# B&R Automation Studio project NewPendant_NG4_11_05_25A (part 22)

##### ArcLink.h
```c
#ifndef _ARCLINK_H
#define _ARCLINK_H

#include <bur/plctypes.h>

#include <runtime.h>

#include <..\..\Lib\utilityLib\bgdebug.h>

#include <..\..\Lib\utilityLib\libRingBuffer.h>

#include <..\..\Lib\arclink\NetworkActions.h>
#include <..\..\Lib\arclink\NetworkAttribute.h>
#include <..\..\Lib\arclink\ArcLinkObject.h>
#include <..\..\Lib\arclink\Robot.h>

#include <..\..\Lib\arclink\WeldController.h>
#include <..\..\Lib\arclink\NetworkBlocks.h>
#include <..\..\Lib\arclink\Attribute.h>

//#include <..\Lib\utilityLib\bgdebug.h>

/*

#include <..\Lib\utilityLib\libRingBuffer.h>

#include <..\Lib\arclink\NetworkActions.h>
#include <..\Lib\arclink\NetworkAttribute.h>
#include <..\Lib\arclink\ArcLinkObject.h>
#include <..\Lib\arclink\Robot.h>

#include <..\Lib\arclink\WeldController.h>
#include <..\Lib\arclink\NetworkBlocks.h>
#include <..\Lib\arclink\Attribute.h>

*/

#define ARC_LINK_OBJECT_BUS_MASTER_ADDRESS 	0
#define ARC_LINK_HEADER_SIZE 				10
#define ARC_LINK_REQUEST_SIZE 				18 // Without Data
#define ARC_LINK_RESPONSE_SIZE 				6 // Without Data

#define ARC_LINK_TXT_BUF_LEN 	512
#define ARC_LINK_TXT_REC_NUM 	8
#define ARC_LINK_TELEMETRY_DESTINATION_ADDRESS 128
#define ACR_LINK_TELEMETRY_ALL_OBJECT_ADDRESS 254

/* Arclink Message  */
typedef struct Arc_Link_Internal_typ{
	UDINT MaxMsgDataLength;
	USINT *pInMsg;
	UDINT  InMsgLen;
	USINT *pOutMsg;
	UDINT  OutMsgLen;

	USINT  InMsgCnt;
	USINT  OutMsgCnt;

} Arc_Link_Internal_typ;

/**
 * @author Obed Bardales
 *         <p>
 *         <b>ArcLink UDP Message Header</b>, which is required in any
 *         ArcLink/XT transmission, has the following structure:
 *         </p>
 *         <br>
 *
 */
typedef struct Arc_Link_Header_typ
{
		/**
	 * <b>Flags</b>: The Flags are a number of boolean settings which control
	 * the type and behavior of the given message packet. (See Table 13 2
	 * Message Header Flags Bit fields) <br>
	 * <b>Value / Range</b>: 0 to 65535 <br>
	 * <b>Size</b>: 2 <i>bytes</i><br>
	 * Bits Description<br>
	 * 0 (LSB) If not set, then the accompanying message is a request. If set,
	 * then the message is a response.<br>
	 * 1 If not set, then the accompanying message is a Server Command. If set,
	 * then the message is an ArcLink Command. ArcLink/XT does not use server
	 * commands; this bit must be set.<br>
	 * 2 Flag for whether Group Addressing is to be used. ArcLink/XT does not
	 * support Group requests; this bit must be cleared.<br>
	 * 3 Flag for whether Sessions should be used. ArcLink/XT does not use
	 * sessions; this bit must be cleared<br>
	 * 13 – 15 3-bit number (0 – 7) indicating the Last Error Type (to accompany
	 * LastError in the Message Header) (See Table 13 3 Error Types) <br>
	 * Table 13 2 Message Header Flags Bit fields <br>
	 * <br>
	 * Error Types<br>
	 * Type Description<br>
	 * 1 Port Error. Occurs in the event of a timeout or a framing error on a
	 * certain port.<br>
	 * 2 NA<br>
	 * 3 Windows Error. Occurs when a COM port fails, or on file access
	 * errors.<br>
	 * 4 Server Error. Occurs in the event of a timeout on the server side, a
	 * malformed ALTCP message, or a bad argument in a server command.<br>
	 * 5 ArcLink Error. Occurs on the ArcLink side only.<br>
	 * 6 WinSock Error. Occurs when a socket is closed unexpectedly. <br>
	 * Table 13 3 Error Types<br>
	 *
	 *
	 */
	UINT Flags;
	/**
	* <b>Sequence</b>: A simple number used to identify the process which
	* initially sent the request. Response should match request. Should not be
	* advanced on a message retry attempt. <br>
	* <b>Value / Range</b>: 0 to 65535 <br>
	* <b>Size</b>: 2 <i>bytes</i>
	*/
	UINT Sequence;
	/**
	 * <b>Last Error</b>: In responses, used to inform the application that an
	 * error occurred while processing the requested command. A value of 0
	 * implies no error. <br>
	 * <b>Value / Range</b>: 0 to 4G<br>
	 * <b>Size</b>: 4 <i>bytes</i>
	 */
	UDINT LastError;
	/**
	* <b>Data Length</b>: The size of the entire message packet, not including
	* this header. <br>
	* <b>Value / Range</b>: 0 to 65535<br>
	* <b>Size</b>: 2 <i>bytes</i>
	*/
	UINT DataLength;
} Arc_Link_Header_typ;

/*
	ArcLink ServiceID
*/
typedef struct ServiceID_typ{
	UINT 	AttributeNumber;
	USINT	StateNumber;
	USINT	PropertyNumber;
} ServiceID_typ;

/**
 * @author Obed Bardales
 *         <p>
 *         <b>ArcLink Requests</b>, If the incoming message is an ArcLink
 *         Command (Bit 1 of the Flags is set), then the data immediately
 *         following the header will be an ArcLink Command Request.
 *         </p>
 *         <br>
 *
 */
typedef struct Arc_Link_Request_typ
{
	/**
	 * <b>Timeout Time (10-ms ticks)</b>: Response time-out time for proxied CAN
	 * requests (default is 100), 20ms recommended.<br>
	 * <b>Value / Range</b>: 0 to 65535 <br>
	 * <b>Size</b>: 2 <i>bytes</i>
	 */
	UINT TimeoutTime;
	/**
	 * <b>Flags</b>: Several boolean settings to further configure the command
	 * request. (See Table 13.5 ArcLink Command Request Flags Bit fields)<br>
	 * <b>Value / Range</b>: 0 to 255 <br>
	 * <b>Size</b>: 1 <i>byte</i> Bits Description <br>
	 * (LSB) 0 - 1 Response Filter Type (0 to 3)<br>
	 * 0 = Match (default)<br>
	 * 1 = First-in<br>
	 * 2 Abort (default is false)<br>
	 * 3 Specifies whether the Timeout Time in the Command Request applies to
	 * each individual response (true) or all responses at once (false).<br>
	 *
	 */
	USINT Flags;
	/**
	 * <b>Retries</b>: Number of retry attempts for proxied CAN requests
	 * (default is 1)<br>
	 * <b>Value / Range</b>: 0 to 255 <br>
	 * <b>Size</b>: 1 <i>byte</i>
	 */
	USINT Retries;

	/**
	 * <b>Message Counter</b>: A simple number used to identify the process
	 * which initially sent the request. Response should match request. Should
	 * not be advanced on a message retry attempt. <br>
	 * <b>Value / Range</b>: 0 to 255 <br>
	 * <b>Size</b>: 1 <i>byte</i>
	 */
	USINT MessageCounter;

	/**
	 * <b>Addressing Mode</b>: Addressing Mode to use (default is peer-peer)
	 * (See Table 13 6 Addressing Modes) ArcLink/XT may not make requests using
	 * group addressing. <br>
	 * <b>Value / Range</b>: 0 to 255 <br>
	 * <b>Size</b>: 1 <i>byte</i><br>
	 * Mode Description <br>
	 * 0 Master-Slave<br>
	 * 1 Master-Slaves<br>
	 * 4 Slave-Master<br>
	 * 6 Peer-Peer<br>
	 * 7 Peer-Peers<br>
	 *
	 */
	USINT AddressingMode;

	/**
	 * <b>Connection ID</b>: Connection ID to use (default is 15) (See Table
	 * 13.7 Connection IDs) <br>
	 * <b>Value / Range</b>: 0 to 255 <br>
	 * <b>Size</b>: 1 <i>byte</i><br>
	 * ID Description<br>
	 * 2 Active Master-Slave<br>
	 * 3 Active Slave-Master Active Peer-Peer<br>
	 * 15 General<br>
	 *
	 */
	USINT ConnectionID;

	/**
	 * <b>Maximum Objs</b>: Maximum number of ArcLink Object respondents. If
	 * Group Addressing is not used, then this value must be set to 1.
	 * ArcLink/XT should set this field to 1. <br>
	 * <b>Value / Range</b>: 0 to 255 <br>
	 * <b>Size</b>: 1 <i>byte</i>
	 */
	USINT MaximumObjs;

	/**
	 * <b>Service ID</b>: (See Attribute Service ID)<br>
	 * <b>Value / Range</b>: ... <br>
	 * <b>Size</b>: 4 <i>bytes</i><br>
	 *
	 * Attributes are referenced using an attribute service ID. Table 15 2 shows
	 * that this structure includes an attribute number, a property number and a
	 * state number. The state is only relevant for attributes whose Attribute
	 * Class Property is set to 10 or 11, in which case the state field selects
	 * the state. If a state is not applicable for the attribute in question,
	 * the value in this field is ignored.<br>
	 *
	 * |Attribute Number| State Number |Attribute Property Number E.g. Value, Low limit, High limit| <br>
	 * |2 bytes |1 byte |1 byte |<br>
	 * Table 15 2- Attribute Service ID
	 *
	 *
	 */
	ServiceID_typ ServiceID;

	/**
	 * <b>Source Address</b>: Source address of the message.<br>
	 * <b>Value / Range</b>: 0 - 255 <br>
	 * <b>Size</b>: 1 <i>byte</i>
	 */
	USINT SourceAddress;

	/**
	 * <b>Destination Address</b>: Destination Address of the message. Either an
	 * ArcLink Object network address or an ArcLink Group Network address,
	 * depending on the Addressing Mode ArcLink/XT may not make requests using
	 * group addressing. <br>
	 * <b>Value / Range</b>: 0 - 255 <br>
	 * <b>Size</b>: 1 <i>byte</i><br>
	 *
	 * <b>24. ArcLink Object Classes</b><br>
	 * Object Object Class Function<br>
	 * Bus Master (BM) 0 Assigns (“maps”) ArcLink addresses.<br>
	 * Weld-Controller (WC) 1 Contains power on/off and welding process
	 * adjustments for the welding power supply.<br>
	 * Wire Drive (WD) 2 Contains motor on/off and set wire feed speed command
	 * value.<br>
	 * User Interface 3 Manual user interface<br>
	 * Gas Controller (GC) 4 Contains the gas on/off command to control the gas
	 * solenoid.<br>
	 * Sense Lead (SL) 5 Controls remote torch voltage electrode sense
	 * connection<br>
	 * DeviceNet Gateway 6 DeviceNet Gateway<br>
	 * Reserved 7 <br>
	 * Ethernet Gateway (GW) 8 Ethernet Gateway. This is the gateway over which
	 * ArcLink/XT messages arrive.<br>
	 * Spool Gun 9 Spool Gun<br>
	 * Robot 10 Controls the other objects.<br>
	 * Phase Generator 11 Phase Generator. In ACDC systems, this determines the
	 * frequency and phase relationships (from arc to arc).<br>
	 * Arc Object 12 The Arc Object is used in previous generation ACDC
	 * systems.<br>
	 * Reserved 13 <br>
	 * Dual User Interface 14 Dual manual feeder user interface.<br>
	 * Pendent 15 Manual operator pendent.<br>
	 * Reserved 16 <br>
	 * Process Monitor 17 The Process Monitor object records welding data and
	 * enforces process limits (if set).<br>
	 * Spread Arc 18 The spread arc device oscillates the welding torch.<br>
	 * Flux Hopper 19 The flux hopper dispenses flux in SAW welding.<br>
	 * Tractor Travel 20 The tractor moves the welding torch.<br>
	 * Travel Carriage 21 The travel carriage moves the welding torch.<br>
	 * Remote 22 The remote reads analog inputs (for remote analog
	 * pendants).<br>
	 * Stick/TIG UI 23 The Stick/TIG UI is a limited function manual user
	 * interface.<br>
	 * STT Switch 24 The STT switch is used in the STT process.<br>
	 * AC Switch 25 The AC switch is used in AC processes.<br>
	 *
	 */
	USINT DestinationAddress;

	/**
	 * <b>Service</b>: Number of the service to execute (See Appendix: Network
	 * Services) <br>
	 * <b>Value / Range</b>: 0 - 255 <br>
	 * <b>Size</b>: 1 <i>byte</i>
	 */
	USINT Service;

	/**
	 * <b>Max Response Size</b>: Maximum size of the response (in bytes) <br>
	 * <b>Value / Range</b>: 0 - 254 <br>
	 * <b>Size</b>: 1 <i>byte</i>
	 */
	USINT MaxResponseSize;

	/**
	 * <b>Request Size</b>: Size of outgoing ArcLink Data<br>
	 * <b>Value / Range</b>: 0 - 255 <br>
	 * <b>Size</b>: 1 <i>byte</i>
	 */
	USINT RequestSize;

	/**
	 * <b>Reserved</b>: A reserved byte<br>
	 * <b>Value / Range</b>: 0 - 255 <br>
	 * <b>Size</b>: 1 <i>byte</i>
	 */
	USINT Reserved;

	/**
	 * <b>OutgoingData</b>: Outgoing ArcLink data<br>
	 * <b>Value / Range</b>: ... <br>
	 * <b>Size</b>: 2+ <i>bytes</i>
	 */

	USINT* OutgoingData;
} Arc_Link_Request_typ;

/**
 * @author Obed Bardales
 *         <p>
 *         <b>ArcLink Response</b>, A response to an ArcLink Command request
 *         coming back from the machine must be preceded by an ALTCP header, as
 *         specified above. The header’s Flags must have bits 0 and 1 set to
 *         True in order to be identified as an ArcLink response. Immediately
 *         after the header, the ArcLink Command Response is structured as
 *         follows
 *         </p>
 *         <br>
 *
 */
typedef struct Arc_Link_Response_typ
{
	/**
	 * <b>Object Count</b>: Number of objects that responded to the ArcLink
	 * request<br>
	 * <b>Value / Range</b>: 0 to 255 <br>
	 * <b>Size</b>: 1 <i>byte</i>
	 */
	USINT ObjectCount;
	/**
	* <b>Reserved</b>: A reserved byte<br>
	* <b>Value / Range</b>: 0 to 255 <br>
	* <b>Size</b>: 1 <i>byte</i>
	*/
	USINT Reserved;
	/**
	 * <b>Status</b>: If the request had caused an ArcLink error, the error will
	 * be recorded in this status byte. If there was no error, status will be
	 * 0.<br>
	 * <b>Value / Range</b>: 0 to 255 <br>
	 * <b>Size</b>: 1 <i>byte</i>
	 */
	USINT Status;
	/**
	 * <b>Object Address</b>: The ArcLink network address of the object that
	 * responded. <br>
	 * <b>Value / Range</b>: 0 to 255 <br>
	 * <b>Size</b>: 1 <i>byte</i>
	 */
	USINT ObjectAddress;
	/**
	 * <b>Response Size</b>: The size (in bytes) of the incoming ArcLink Data
	 * <br>
	 * <b>Value / Range</b>: 0 to 254 <br>
	 * <b>Size</b>: 1 <i>byte</i>
	 */
	USINT ResponseSize;
	/**
	 * <b>Reserved</b>: A reserved byte<br>
	 * <b>Value / Range</b>: 0 to 255 <br>
	 * <b>Size</b>: 1 <i>byte</i>
	 */
	USINT Reserved2;
	/**
	 * <b>Response Data</b>: Incoming ArcLink Data<br>
	 * <b>Value / Range</b>: ... <br>
	 * <b>Size</b>: 2+ <i>bytes</i>
	 */
	USINT* ResponseData;
} Arc_Link_Response_typ;

/* Arclink Message  */
typedef struct Arc_Link_Message_typ{
	Arc_Link_Header_typ header;
	Arc_Link_Request_typ request;
	Arc_Link_Response_typ response;
} Arc_Link_Message_typ;

typedef struct PendingResponse_typ{
	BOOL WriteAttribute30770;   //1 Enable
	BOOL WriteAttribute30781;   //1 Enable
	BOOL WriteAttribute30758;   //1 Enable
	BOOL WriteAttribute30;
	BOOL CreateReadyReport;
	BOOL CreateFaultReport;

	UINT fsSequence;  // Sequence tracked for attribute 30731 (fault status)
	UINT sqConfigDataSearchAction;
	UINT sqReadCoolerSens;
	UINT WriteAttribute30770Sequence;
	UINT WriteAttribute30781Sequence;
	UINT WriteAttribute30758Sequence;
	UINT WriteAttribute30Sequence;
	UINT CreateReadyReportSequence;
	UINT CreateFaultReportSequence;
	UINT CreateReadControlParamDataAction;
	UINT sqConfigDataSearchAction_GasSol;

} PendingResponse_typ;

typedef struct Arc_Link_typ
{
	RingBuffer *bufIN; 		// Incoming Messages RingBuffer pointer
	RingBuffer *bufOUT; 	// Outgoing Messages RingBuffer pointer
	Arc_Link_Message_typ msgIN;		// Placeholder
	Arc_Link_Message_typ msgOUT;	// Placeholder
	Arc_Link_Internal_typ internal; // Internal
	Robot_typ robot; // Robot reference to this plc
	PendingResponse_typ PendingResponse; // pending response
} Arc_Link_typ;

/* Prototypes */
void ArcLink_cyclic(Arc_Link_typ *arc);
void ArcLink_init(Arc_Link_typ *arc , RingBuffer *bufIN, RingBuffer *bufOUT , UDINT  pInMsg  , UDINT  pOutMsg , UDINT recLen );

//////////////////////////////////////////////////////////////////////
// ArcLink Event Codes
// The following table lists the event codes that can be logged in Event Log postings
//////////////////////////////////////////////////////////////////////
#define	ARC_LINK_EVENT_11	11	/* 	Internal request failed to generate a response */
#define	ARC_LINK_EVENT_12	12	/* 	Internal attribute read/write failed */
#define	ARC_LINK_EVENT_13	13	/* 	Values/settings saved in the system could not be restored (corrupt)*/
#define	ARC_LINK_EVENT_14	14	/* 	Values/settings saved in the system could not be restored (primary section) */
#define	ARC_LINK_EVENT_15	15	/* 	Values/settings saved in the system could not be restored (secondary section) */
#define	ARC_LINK_EVENT_16	16	/* 	Values/settings that are saved could not be restored during powerup */
#define	ARC_LINK_EVENT_17	17	/* 	Serial port communication timed out*/
#define	ARC_LINK_EVENT_18	18	/* 	ArcLink auto-mapping failed*/
#define	ARC_LINK_EVENT_19	19	/* 	Excessive EEPROM saves detected for a certain attribute */
#define	ARC_LINK_EVENT_21	21	/* 	Device that controls sequence of the welding operation halted due to an error*/
#define	ARC_LINK_EVENT_22	22	/* 	Device that controls the sequence of the welding operation halted due to an error response when it tried to update a device's settings*/
#define	ARC_LINK_EVENT_23	23	/* 	Weld Sequencer could not change settings on a controlled object during welding*/
#define	ARC_LINK_EVENT_24	24	/* 	Error occurred while the weld sequencer was changing the weld mode*/
#define	ARC_LINK_EVENT_25	25	/* 	When updating non-state memory attributes via sequencer action, allow all but mode changing*/
#define	ARC_LINK_EVENT_26	26	/* 	Problem with paired mapping*/
#define	ARC_LINK_EVENT_27	27	/* 	Read/write request failed during paired mapping*/
#define	ARC_LINK_EVENT_28	28	/* 	Output locked out in the Weld Controller*/
#define	ARC_LINK_EVENT_29	29	/* 	Low-level DSP main control routine could not complete all of its tasks in time*/
#define	ARC_LINK_EVENT_31	31	/* 	Actual input current exceeded the input current limit*/
#define	ARC_LINK_EVENT_32	32	/* 	Capacitor bank A fell below the low voltage limit*/
#define	ARC_LINK_EVENT_33	33	/* 	Capacitor bank B fell below the low voltage limit*/
#define	ARC_LINK_EVENT_34	34	/* 	Capacitor bank A exceeded the high voltage limit*/
#define	ARC_LINK_EVENT_35	35	/* 	Capacitor bank B exceeded the high voltage limit*/
#define	ARC_LINK_EVENT_36	36	/* 	System detected a temperature level beyond the normal system operating limit*/
#define	ARC_LINK_EVENT_37	37	/* 	System failed to initialize inverter hardware during startup*/
#define	ARC_LINK_EVENT_38	38	/* 	Momentary AC dropout*/
#define	ARC_LINK_EVENT_39	39	/* 	Miscellaneous hardware fault occurred whose source cannot be determined*/
#define	ARC_LINK_EVENT_41	41	/* 	Long-term average secondary (weld) current limit has been exceeded*/
#define	ARC_LINK_EVENT_42	42	/* 	System detected a ground fault has occurred*/
#define	ARC_LINK_EVENT_43	43	/* 	Voltage difference between Capacitor bank A and B was greater than the allowable limit*/
#define	ARC_LINK_EVENT_44	44	/* 	Main processor in the system did not respond to another processor within the allotted time*/
#define	ARC_LINK_EVENT_45	45	/* 	Welding voltage was above limit*/
#define	ARC_LINK_EVENT_46	46	/* 	Output amperage limit exceeded*/
#define	ARC_LINK_EVENT_47	47	/* 	Miscellaneous hardware fault (capacitor fault or heart beat fault)*/
#define	ARC_LINK_EVENT_48	48	/* 	Miscellaneous hardware fault (main contactor open)*/
#define	ARC_LINK_EVENT_49	49	/* 	Single phase input operation has been detected*/
#define	ARC_LINK_EVENT_51	51	/* 	Weld Controller failed to set weld sequencer schedule memory*/
#define	ARC_LINK_EVENT_52	52	/* 	Digital Signal Processor (DSP) in the system is no longer responding to heartbeat request from the main processor*/
#define	ARC_LINK_EVENT_53	53	/* 	System detected the loss of a voltage sense lead*/
#define	ARC_LINK_EVENT_54	54	/* 	Long-term average secondary (weld) current limit has been exceeded*/
#define	ARC_LINK_EVENT_55	55	/* 	Communication with DSP failed*/
#define	ARC_LINK_EVENT_56	56	/* 	Communication with Chopper failed*/
#define	ARC_LINK_EVENT_57	57	/* 	Function Generator reported an error*/
#define	ARC_LINK_EVENT_58	58	/* 	Primary input power board not ready*/
#define	ARC_LINK_EVENT_59	59	/* 	Reduced input power detected*/
#define	ARC_LINK_EVENT_61	61	/* 	Step value for either upslope or downslope was calculated to zero*/
#define	ARC_LINK_EVENT_62	62	/* 	Weld Sequencer did not get a positive response after sending out Weld Cycle Data twice*/
#define	ARC_LINK_EVENT_63	63	/* 	Problem with submerged arc Slave device*/
#define	ARC_LINK_EVENT_71	71	/* 	Secondary over-power*/
#define	ARC_LINK_EVENT_72	72	/* 	Unsupported hardware revision*/
#define	ARC_LINK_EVENT_81	81	/* 	Feed head experienced a motor overload fault*/
#define	ARC_LINK_EVENT_82	82	/* 	Feed head experienced a motor over current fault*/
#define	ARC_LINK_EVENT_83	83	/* 	Wire drive shutdown bit 1 circuit open*/
#define	ARC_LINK_EVENT_84	84	/* 	Wire drive shutdown bit 2 circuit open (Water Fault)*/
#define	ARC_LINK_EVENT_85	85	/* 	Object could not find the Arc Control Object to send the I/O trigger command*/
#define	ARC_LINK_EVENT_86	86	/* 	Wire Drive input voltage too high*/
#define	ARC_LINK_EVENT_87	87	/* 	Wire Drive failed to find another object*/
#define	ARC_LINK_EVENT_88	88	/* 	Wire Drive could not send the trigger to the specified object in the event data.*/
#define	ARC_LINK_EVENT_89	89	/* 	Wire Drive failed to find the Production Monitoring object for profile selection based on digital inputs*/
#define	ARC_LINK_EVENT_91	91	/* 	Sense Lead object could not update the weld sequencer's or the weld controller's polarity attribute.*/
#define	ARC_LINK_EVENT_92	92	/* 	Remote shutdown of Weld Controller*/
#define	ARC_LINK_EVENT_95	95	/* 	Spool Gun shutdown due to motor drawing excessive current*/
#define	ARC_LINK_EVENT_96	96	/* 	Weld Controller failed to read WFS decimal places*/

//////////////////////////////////////////////////////////////////////
// ArcLink Error Codes
// The following table lists the event codes that can be logged in Event Log postings
//////////////////////////////////////////////////////////////////////
#define	ARC_LINK_ERROR_0	0	/*	Success (no message error). */
#define	ARC_LINK_ERROR_1  	1	/*	Attribute not found. */
#define ARC_LINK_ERROR_2	2	/* 	Attribute value is read-only. */
#define ARC_LINK_ERROR_3	3 	/* 	Attribute Value (being written) is out of limits.*/
#define ARC_LINK_ERROR_4	4	/* 	Attribute Value (being written) is above high limit.*/
#define ARC_LINK_ERROR_5	5	/* 	Attribute Value (being written) is below low limit.*/
#define ARC_LINK_ERROR_8	8	/*	ArcLink object not found (bad ArcLink object address).*/
#define ARC_LINK_ERROR_9	9	/*	Attribute property specified is invalid.*/
#define ARC_LINK_ERROR_11	11	/*	Attribute property is not applicable (e.g. units code for Boolean type).  Only while reading.*/
#define ARC_LINK_ERROR_12	12	/*	Attribute property is not supported (e.g. invalid type id, or not applicable).  For reads or writes.*/
#define ARC_LINK_ERROR_13	13	/*	Attribute property is read-only.*/
#define ARC_LINK_ERROR_14	14	/*	Attribute is invalid.*/
#define ARC_LINK_ERROR_15	15	/*	ArcLink Object messages could not be relayed over Ethernet.*/
#define ARC_LINK_ERROR_16 	16	/*	ArcLink service busy (message should be re-sent).*/
#define ARC_LINK_ERROR_17	17	/*	ArcLink service busy (message should be re-sent).*/
#define ARC_LINK_ERROR_18	18	/*	ArcLink service busy (message should be re-sent).*/
#define ARC_LINK_ERROR_20	20	/*	ArcLink Block ID not found (for block read or write service).*/
#define ARC_LINK_ERROR_21	21	/*	ArcLink Action ID not found (for action service).*/
#define ARC_LINK_ERROR_22	22	/*	ArcLink Group Address not found.*/
#define ARC_LINK_ERROR_23	23	/*	ArcLink Event ID not found.*/
#define ARC_LINK_ERROR_24	24	/*	ArcLink Service not supported.*/
#define ARC_LINK_ERROR_25	25	/*	ArcLink Service not available.*/
#define ARC_LINK_ERROR_26	26	/*	Fragment buffer busy (message should be re-sent).*/
#define ARC_LINK_ERROR_27	27	/*	Fragment out of sequence (message should be re-started).*/
#define ARC_LINK_ERROR_28	28	/*	Fragment receive time out (message should be re-started).*/
#define ARC_LINK_ERROR_29	29	/*	Fragment message invalid.*/
#define ARC_LINK_ERROR_30	30	/*	Message request size is invalid.*/
#define ARC_LINK_ERROR_31	31	/*	Message response buffer was too small.*/
#define ARC_LINK_ERROR_33	33	/*	Message time out (message should be re-started).*/
#define ARC_LINK_ERROR_34	34	/*	Write failed.*/
#define ARC_LINK_ERROR_35	35	/*	Read failed.*/
#define	ARC_LINK_ERROR_36	36	/*	Invalid selection.*/
#define	ARC_LINK_ERROR_37	37	/*	ArcLink Object was busy (message should be re-sent). */

//////////////////////////////////////////////////////////////////////
// Attribute Value Property ID Codes
//////////////////////////////////////////////////////////////////////
/*
 * Value 0 Defined by Attribute Data Type
 */
#define PROPERTY_ID_VALUE 0

/**
 * Class 1 Unsigned Int (1)
 */
#define PROPERTY_ID_CLASS 1

/**
 * Saved In E2 2 Boolean
 */
#define PROPERTY_ID_SAVED_IN_E2 2

/**
 * Attribute Data Type 3 Unsigned Int (1)
 */
#define PROPERTY_ID_ATTRIBUTE_DATA_TYPE 3

/**
 * Unit Code 4 Unsigned Int (1)
 */
#define PROPERTY_ID_UNIT_CODE 4

/**
 * High Limit 5 Defined by Attribute Data Type
 */
#define PROPERTY_ID_HIGH_LIMIT 5

/**
 * Low Limit 6 Defined by Attribute Data Type
 */
#define PROPERTY_ID_LOW_LIMIT 6

/**
 * Decimal Places 7 Unsigned Int (1)
 */
#define PROPERTY_ID_DECIMAL_PLACES 7

/**
 * Name 8 String (1-254)
 */
#define PROPERTY_ID_NAME 8

//////////////////////////////////////////////////////////////////////
// Attribute Data Type Property, ID Codes
//////////////////////////////////////////////////////////////////////
/**
 * <b>Boolean</b>:<br>
 * <i>size: 1 byte</i>
 */
#define DATA_TYPE_BOOLEAN 0

/**
 * <b>Enumerated 1</b>:<br>
 * <i>size: 1 byte</i>
 */
#define DATA_TYPE_ENUMERATED_1 1

/**
 * <b>Enumerated 2</b>:<br>
 * <i>size: 2 bytes</i>
 */
#define DATA_TYPE_ENUMERATED_2 2

/**
 * <b>Enumerated 4</b>:<br>
 * <i>size: 4 bytes</i>
 */
#define DATA_TYPE_ENUMERATED_4 3

/**
 * <b>Bit Mapped 1</b>:<br>
 * <i>size: 1 byte</i>
 */
#define DATA_TYPE_BIT_MAPPED_1 4

/**
 * <b>Bit Mapped 2</b>:<br>
 * <i>size: 2 bytes</i>
 */
#define DATA_TYPE_BIT_MAPPED_2 5

/**
 * <b>Bit Mapped 4</b>:<br>
 * <i>size: 4 bytes</i>
 */
#define DATA_TYPE_BIT_MAPPED_4 6

/**
 * <b>Signed Integer 1</b>:<br>
 * <i>size: 1 byte</i>
 */
#define DATA_TYPE_SIGNED_INTEGER_1 7

/**
 * <b>Signed Integer 2</b>:<br>
 * <i>size: 2 bytes</i>
 */
#define DATA_TYPE_SIGNED_INTEGER_2 8

/**
 * <b>Signed Integer 4</b>:<br>
 * <i>size: 4 bytes</i>
 */
#define DATA_TYPE_SIGNED_INTEGER_4 9

/**
 * <b>Unsigned Integer 1</b>:<br>
 * <i>size: 1 byte</i>
 */
#define DATA_TYPE_UNSIGNED_INTEGER_1 10

/**
 * <b>Unsigned Integer 2</b>:<br>
 * <i>size: 2 bytes</i>
 */
#define DATA_TYPE_UNSIGNED_INTEGER_2 11

/**
 * <b>Unsigned Integer 4</b>:<br>
 * <i>size: 4 bytes</i>
 */
#define DATA_TYPE_UNSIGNED_INTEGER_4 12

/**
 * <b>Floating Point</b>:<br>
 * <i>size: 4 bytes</i>
 */
#define DATA_TYPE_FLOATING_POINT 13

/**
 * <b>ASCII String </b>:<br>
 * <i>size: (0 - 254) bytes</i>
 */
#define DATA_TYPE_ASCII_STRING 14

//////////////////////////////////////////////////////////////////////
// Attribute Class Codes
//////////////////////////////////////////////////////////////////////
/**
 * <b>Network Configuration</b>:<br>
 * Inputs related to the network. E.g. Group Assignment <br>
 *
 */
#define CLASS_NETWORK_CONFIGURATION 0

/**
 * <b>Network Status</b>:<br>
 * Outputs describing information related to the network. E.g. Network
 * Version Number <br>
 * <i>Read Only</i>
 */
#define CLASS_NETWORK_STATUS 1

/**
 * <b>Command</b>:<br>
 * Inputs used to activate an object?s behavior. Changes generally have an
 * immediate effect. E.g. Gas Purge<br>
 *
 */
#define CLASS_COMMAND 2

/**
 * <b>Reference</b>:<br>
 * Inputs which are set points. Changes generally have an immediate effect.
 * E.g. Cold Inch<br>
 *
 */
#define CLASS_REFERENCE 3

/**
 * <b>Reference</b>:<br>
 * Inputs which alter the object?s general behavior. E.g. Motor Control-Loop
 * Mode<br>
 *
 */
#define CLASS_CONFIGURATION 4

/**
 * <b>Signal</b>:<br>
 * Outputs used for metering and monitoring. E.g. Actual Arc Current <br>
 * <i>Read Only</i>
 */
#define CLASS_SIGNAL 5

/**
 * <b>Status</b>:<br>
 * Outputs used for metering and monitoring. E.g. Faults<br>
 * <i>Read Only</i>
 */
#define CLASS_STATUS 6

/**
 * <b>Sequence Controlled Command</b>:<br>
 * Command to be controlled by the Sequencer object (object class 0). E.g.
 * Motor On/Off<br>
 */
#define CLASS_SEQUENCE_CONTROLLED_COMMAND 7

/**
 * <b>Sequence Controlled Reference</b>:<br>
 * Reference to be controlled by the Sequencer object (object class 0). E.g.
 * Commanded WFS<br>
 */
#define CLASS_SEQUENCE_CONTROLLED_REFERENCE 8

/**
 * <b>Sequence Controlled Configuration</b>:<br>
 * Configuration to be controlled by the Sequencer object (object class 0).
 * E.g. Weld Procedure <br>
 */
#define CLASS_SEQUENCE_CONTROLLED_CONFIGURATION 9

/**
 * <b>Command with State Memory</b>:<br>
 * Command which has state memory. The sequencer object creates attributes
 * of this class from attributes of class 7. The state portion of the
 * service ID is relevant for the read and write services.<br>
 */
#define CLASS_COMMAND_WITH_STATE_MEMORY 10

/**
 * <b>Reference with State Memory</b>:<br>
 * Reference which has state memory. The sequencer object creates attributes
 * of this class from attributes of class 8. The state portion of the
 * service ID is relevant for the read and write services.<br>
 */
#define CLASS_REFERENCE_WITH_STATE_MEMORY 11

/**
 * <b>Debug</b>:<br>
 * Used (primarily) during manufacturing.
 */
#define CLASS_DEBUG 12

/**
 * <b>Setup</b>:<br>
 */
#define CLASS_SETUP 13

/**
 * <b>Version</b>:<br>
 * Version related information.<br>
 * <i>Read Only</i>
 */
#define CLASS_VERSION 14

//////////////////////////////////////////////////////////////////////
// Addresing mode
//////////////////////////////////////////////////////////////////////
#define ADDRESS_MODE_MASTER_SLAVE	 0
#define ADDRESS_MODE_MASTER_SLAVES	 1
#define ADDRESS_MODE_SLAVE_MASTER	 4
#define ADDRESS_MODE_PEER_PEER		 6
#define ADDRESS_MODE_PEER_PEERS 	 7

//////////////////////////////////////////////////////////////////////
// Network Services Codes
//////////////////////////////////////////////////////////////////////
/**
 * <b>Attribute Read</b>:<br>
 */
#define NETWORK_SERVICE_ATTRIBUTE_READ 0

/**
 * <b>Attribute Write</b>:<br>
 */
#define NETWORK_SERVICE_ATTRIBUTE_WRITE 1

/**
 * <b>Confirmed Event Report</b>:<br>
 */
#define NETWORK_SERVICE_CONFIRMED_EVENT_REPORT 2

/**
 * <b>Unconfirmed Event Report</b>:<br>
 */
#define NETWORK_SERVICE_UNCONFIRMED_EVENT_REPORT 3

/**
 * <b>Action</b>:<br>
 */
#define NETWORK_SERVICE_ACTION 4

/**
 * <b>Read Block</b>:<br>
 */
#define NETWORK_SERVICE_READ_BLOCK 5

/**
 * <b>Write Block</b>:<br>
 */
#define NETWORK_SERVICE_WRITE_BLOCK 6

/**
 * <b>Confirmed Event Block Report</b>:<br>
 */
#define NETWORK_SERVICE_CONFIRMED_EVENT_BLOCK_REPORT 7

/**
 * <b>Unconfirmed Event Block Report</b>:<br>
 */
#define NETWORK_SERVICE_UNCONFIRMED_EVENT_BLOCK_REPORT 8

//#include <..\..\Lib\arclink\Handler.h>

#endif /* _ARCLINK_H */
```

##### Robot.c
```c
/*
 * Handler.c
 *
 *  Created on: May 18, 2017
 *      Author: Obed Bardales
 */
#ifndef _ROBOT_C
#define _ROBOT_C

/* Handle Robot Cyclic Operations */
void handleRobotCyclicOps(Arc_Link_typ *arc){
	if(!arc) return;

	// Handle Mr.Robot interface
	handleRobotInterface(arc);

	// "The difference is not one thing, it's everything!"
}

/* Get Network Configuration from Robot */
void getNetworkConfigurationAttribute(Arc_Link_typ *arc, USINT *ResponseData){
	Arc_Link_Request_typ *req;
	Arc_Link_Response_typ *r;
	Robot_typ *robot;
	ServiceID_typ *serviceID;
	ArcLinkObject_typ *arclink;
	USINT data[10]; // Temp Data place holder
	UINT txtlength; // text length

	if(!arc) return;
	if(!ResponseData) return;

	robot = &arc->robot; // Reference to Robot
	req = &arc->msgIN.request;
	serviceID = &req->ServiceID;
	r = &arc->msgOUT.response;
	arclink = &robot->arclink;
	int dataSize = req->MaxResponseSize;

	/* Attribute Number */
	switch (serviceID->AttributeNumber) {

		case VENDOR_ID: /* 0 */
			// MaxDataSize = 2
			// Big Endian Format

			data[0] = (USINT) (arclink->network.VendorID >> 8);
			data[1] = (USINT) (arclink->network.VendorID >> 0);
			memcpy(ResponseData, data, 2);
			r->ResponseSize = 2;

			return;

		case CLASS_ID: /* 4 */
			// MaxDataSize = 2
			// Big Endian Format
			data[0] = (USINT) (arclink->network.ClassID >> 8);
			data[1] = (USINT) (arclink->network.ClassID >> 0);
			memcpy(ResponseData, data, 2);
			r->ResponseSize = 2;
			return;

		case CLASS_TYPE: /* 7 */
			// MaxDataSize = 2
			// Big Endian Format
			data[0] = (USINT) (arclink->network.ClassType >> 0);
			memcpy(ResponseData, data, 1);
			r->ResponseSize = 1;
			return;

		case GROUP_ASSIGNMENTS: /* 10 */
			// MaxDataSize = 2
			// Big Endian Format
			data[0] = (USINT) (arclink->network.GroupAssignments >> 0);
			memcpy(ResponseData, data, 1);
			r->ResponseSize = 1;
			return;

		case INSTANCE_ASSIGNMENTS: /* 11 */
			// MaxDataSize = 2
			// Big Endian Format
			data[0] = (USINT) (arclink->network.InstanceAssignments >> 0);
			memcpy(ResponseData, data, 1);
			r->ResponseSize = 1;
			return;

		case FAULT_STATUS: /* 14 */
			// MaxDataSize = 2
			// Big Endian Format
			data[0] = (USINT) (arclink->network.FaultStatus >> 0);
			memcpy(ResponseData, data, 1);
			r->ResponseSize = 1;
			return;

		case SILICON_SERIAL_NUMBER: /* 16 */
			// MaxDataSize = 2
			// Big Endian Format
			data[0] = (USINT) (arclink->network.SiliconSerialNumber >> 8);
			data[1] = (USINT) (arclink->network.SiliconSerialNumber >> 0);
			memcpy(ResponseData, data, 2);
			r->ResponseSize = 2;
			return;

		case NUMBER_OF_EMBEDDED_OBJECTS: /* 17 */
			// MaxDataSize = 2
			// Big Endian Format
			data[0] = (USINT) (arclink->network.NumberofEmbeddedObjects >> 0);
			memcpy(ResponseData, data, 1);
			r->ResponseSize = 1;
			return;

		case SOFTWARE_VERSION: /* 19 */
			// MaxDataSize = 64
			// Big Endian Format
			txtlength = strlen(arclink->network.SoftwareVersion);
			// Swap Bytes before sendSuccesfullWriteAttributeConfirmation
			//swapBytes(arclink->network.SoftwareVersion, txtlength);
			memcpy(ResponseData, arclink->network.SoftwareVersion, txtlength);
			//swapBytes(arclink->network.SoftwareVersion, txtlength);
			r->ResponseSize = txtlength;
			return;

		case BOOTSTRAP: /* 24 */
			// MaxDataSize = 2
			// Big Endian Format
			data[0] = (USINT) (arclink->network.Bootstrap >> 0);
			memcpy(ResponseData, data, 1);
			r->ResponseSize = 1;
			return;

		case PAIRED_ITEMS_COUNT: /* 50 */
			// MaxDataSize = 2
			// Big Endia Format
			data[0] = (USINT) (arclink->network.PairedItemsCount >> 8);
			data[1] = (USINT) (arclink->network.PairedItemsCount >> 0);
			memcpy(ResponseData, data, 2);
			r->ResponseSize = 2;
			return;
	}
}

/* Write Network Configuration Attribute */
BOOL writeNetworkConfigurationAttribute(Arc_Link_typ *arc){

	BOOL success = 1;

	UINT *data;

	Arc_Link_Request_typ *req;
	ServiceID_typ *serviceID;
	Robot_typ *robot;
	ArcLinkObject_typ *arclink;
	if(!arc) return;

	req = &arc->msgIN.request;
	serviceID = &req->ServiceID;
	robot = &arc->robot;
	arclink = &robot->arclink;

	DBG("Inside writeNetworkConfigurationAttribute \r\n" );
	//Log.d(TAG, "Recevied Assign Network Address Action");

	// Copy Data if available to the Incoming data pointer
	if(req->RequestSize > 0){
	//byte[] data = r.OutgoingData; // incominng data in Big endian format
		data = (arc->internal.pInMsg + ARC_LINK_HEADER_SIZE + ARC_LINK_REQUEST_SIZE); // Pointer to data
	}else{
		DBG("Error: writeNetworkConfigurationAttribute, Error with Request size\r\n" );
		return;
	}

	/* Attribute Number */
	switch (serviceID->AttributeNumber) {

	// Currently Supported Attributes by the Robot
	case RESET:
		arclink->network.Reset = *(data + 0);//data[0]; // Size is typically 1 byte
		arclink->network.BusAvailable = 0; // Robot must enter to unmapped state
		robot->isMapping = 0;
		robot->isMapped = 0;
		robot->Cntrl.Fbk.Status &= ~ArcLink_Mapped;
		robot->Cntrl.Fbk.Status &= ~ArcLink_Mapping;
		robot->isMiscSetupOneShot = 0;
		DBG("Setting Robot to Unmapped state\r\n" );
		break;

	case GROUP_ASSIGNMENTS:
		arclink->network.GroupAssignments = *(data + 0);///data[0]; // Size is typically 1
													// byte

		break;

	case INSTANCE_ASSIGNMENTS:
		arclink->network.InstanceAssignments = *(data + 0);///data[0]; // Size is typically
														// 1 byte
		break;

	case BUS_AVAILABLE:
		arclink->network.BusAvailable = *(data + 0); //data[0]; // Size is typically 1 byte
		robot->isMapping 	= 0;
		robot->isMapped 	= 1;
		robot->Cntrl.Fbk.Status |= ArcLink_Mapped;
		robot->Cntrl.Fbk.Status &= ~ArcLink_Mapping;
		DBG("Robot was mapped succesfully Świetny programista! \r\n" );
		log_event(&robot->eventlog , "Arc Link Mapped");
		break;

	}

	return success; // Whether Attribute was written succesfully

}

void handleRobotInterface(Arc_Link_typ *arc){

	Robot_typ *robot;
	Robot_Intrf_typ *intrf;
	if(!arc) return;

	robot = &arc->robot;
	intrf = &robot->Intrf;

	// Robot must be Mapped with WeldController
	if(!robot->isMapped) return;

	//  Handle state changes from outside and provide feedback

	handleRobotCntrl(arc);
	error_status_handler(arc);
	ArcLink_Timer(arc);
	/////////

	// Handle xCMD
	switch(intrf->xCMD) {
		/* Turn Power Supply ON */
		case ROBOT_CMD_PS_ON:
			writeOutputOnCommand(arc);
			DBG("Robot commanded Power Supply ON! \r\n" );
			log_event(&robot->eventlog , "PS ON Cmd");
			break;

		/* Turn Power Supply OFF */
		case ROBOT_CMD_PS_OFF:
			writeOutputOffCommand(arc);
			DBG("Robot commanded Power Supply OFF! \r\n" );
			log_event(&robot->eventlog , "PS OFF Cmd");
			break;

		/* Set Controls Action Request */
		case ROBOT_SET_CONTROLS:
			createSetControlsAction(arc);
			DBG("Robot sent Set Controls Action Request! \r\n" );
			break;

		case ROBOT_CMD_COOLER_ON:
			writeOutputCoolerOnCommand(arc);
			DBG("Robot commanded Cooler ON! \r\n" );

		break;

		case ROBOT_CMD_COOLER_OFF:
			writeOutputCoolerOffCommand(arc);
			DBG("Robot commanded Cooler OFF! \r\n" );

		break;

		case ROBOT_CMD_SEARCH_COOLER_ADR:
			action_ConfigDataSearch_Cooler(arc);
			DBG("commanded Get Cooler Adr! \r\n" );
		break;

		case ROBOT_READ_COOLER_SENS:
			readAttribute_CoolerSens(arc);
			DBG("commanded Get Cooler Sens! \r\n" );
		break;

		case ROBOT_READ_WC_PARAM_DATA:
			createReadCntrlParamDataAction(arc);
			DBG("commanded Read WC Param Data! \r\n" );
		break;

		case ROBOT_CMD_SEARCH_GAS_SOL_ADR:
			action_ConfigDataSearch_GasSol(arc);
			DBG("commanded Get Gas Sol  Adr! \r\n" );
		break;

		case ROBOT_CMD_GAS_SOL_ENABLE: // Make  Gas Sol “Manual Valve”

			writeOutputGasEnableCommand(arc);
			DBG("Robot commanded Gas Enable\r\n" );

		break;

		case ROBOT_CMD_GAS_SOL_ON: // Turn On Gas Sol

			writeOutputGasOnCommand(arc);
			DBG("Robot commanded Gas ON\r\n" );

		break;

		case ROBOT_CMD_GAS_SOL_OFF:	// Turn Off Gas Sol

			writeOutputGasOffCommand(arc);
			DBG("Robot commanded Gas OFF\r\n" );

		break;

	}

	// Clear xCMD
	if (intrf->xCMD > 0) intrf->xCMD = 0;

}

void handleRobotCntrl(Arc_Link_typ *arc){

	Robot_typ *robot;
	Robot_Intrf_typ *intrf;
	if(!arc) return;

	robot = &arc->robot;
	intrf = &robot->Intrf;

	//*************** CMD  *****************************/
	//**************Highest priority CMD****************//
	if(robot->Cntrl.Cmd.COOLER && !robot->Cntrl.Int._COOLER){

		intrf->xCMD = ROBOT_CMD_COOLER_ON;
		robot->Cntrl.Int._COOLER  = robot->Cntrl.Cmd.COOLER;

	}
	else if(robot->Cntrl.Cmd.RUN != robot->Cntrl.Int._RUN){

		if(robot->Cntrl.Cmd.RUN)
			intrf->xCMD = ROBOT_CMD_PS_ON;
		else
			intrf->xCMD = ROBOT_CMD_PS_OFF;

		robot->Cntrl.Int._RUN  = robot->Cntrl.Cmd.RUN;
	}
	else if(!robot->Cntrl.Cmd.COOLER && robot->Cntrl.Int._COOLER){

		intrf->xCMD = ROBOT_CMD_COOLER_OFF;
		robot->Cntrl.Int._COOLER  = robot->Cntrl.Cmd.COOLER;

	}
	//robot->Cntrl.Int._RUN  = robot->Cntrl.Cmd.RUN;
	//robot->Cntrl.Int._COOLER  = robot->Cntrl.Cmd.COOLER;

	//********************************************************//

	if(!intrf->xCMD){

		/*
		1 Byte	Parameter Mask
		2 Bytes	Weld Mode 	If parameter mask bit 0 set.
		2 Bytes	Work-point	If parameter mask bit 1 set.
		2 Bytes	Trim	If parameter mask bit 2 set.
		2 Bytes	Wave-Control 1	If parameter mask bit 3 set.
		2 Bytes	Wave-Control 2	If parameter mask bit 4 set.
		2 Bytes	Wave-Control 3	If parameter mask bit 5 set.
		2 Bytes	Wave-Control 4	If parameter mask bit 6 set.
		*/

		switch(robot->Cntrl.Cmd.Mode){

			case 3:

				if((robot->Cntrl.Cmd.Mode != robot->Cntrl.Int._Mode )
					|| (robot->Cntrl.Cmd.AmpSP != robot->Cntrl.Int._AmpSP )
					|| (robot->Cntrl.Cmd.BckAmpSP != robot->Cntrl.Int._BckAmpSP )
					|| (robot->Cntrl.Cmd.PulseFreq != robot->Cntrl.Int._PulseFreq )
					|| (robot->Cntrl.Cmd.PulseWidth != robot->Cntrl.Int._PulseWidth )){

					robot->wc.setup.ctrlParam.ParameterMask = 0x23; // 0b0100011; // change accordingly for Mode 3
					UINT *mode 	= &robot->Cntrl.Cmd.Mode; // Mode
					UINT ampSP = (UINT)robot->Cntrl.Cmd.AmpSP; //amps
					robot->wc.setup.ctrlParam.WeldMode = *mode;
					robot->wc.setup.ctrlParam.WorkPoint = ampSP;
					robot->wc.setup.ctrlParam.WaveControl3 = 1; // Hot pulse. Need info from Lincoln

					// This command write Controls Parameter into Power Supply
					intrf->xCMD = ROBOT_SET_CONTROLS;

				}

				robot->Cntrl.Int._Mode 			= robot->Cntrl.Cmd.Mode;
				robot->Cntrl.Int._AmpSP 		= robot->Cntrl.Cmd.AmpSP;
				robot->Cntrl.Int._BckAmpSP 		= robot->Cntrl.Cmd.BckAmpSP;
				robot->Cntrl.Int._PulseFreq 	= robot->Cntrl.Cmd.PulseFreq;
				robot->Cntrl.Int._PulseWidth 	= robot->Cntrl.Cmd.PulseWidth;

			break;

			case 5:

				if((robot->Cntrl.Cmd.Mode != robot->Cntrl.Int._Mode )
					|| (robot->Cntrl.Cmd.Volts != robot->Cntrl.Int._Volts )
					|| (robot->Cntrl.Cmd.Pinch != robot->Cntrl.Int._Pinch )
					){

					robot->wc.setup.ctrlParam.ParameterMask = 0x0D; // 0b0001011; // change accordingly for Mode 5
					UINT *mode 	= &robot->Cntrl.Cmd.Mode; // Mode
					UINT VoltsSP = (UINT)(robot->Cntrl.Cmd.Volts * 10); //Volts
					robot->wc.setup.ctrlParam.WeldMode = *mode;
					robot->wc.setup.ctrlParam.WorkPoint = VoltsSP;
					robot->wc.setup.ctrlParam.WaveControl1 = (UINT)(robot->Cntrl.Cmd.Pinch * 10);

					// This command write Controls Parameter into Power Supply
					intrf->xCMD = ROBOT_SET_CONTROLS;

				}

				robot->Cntrl.Int._Mode 			= robot->Cntrl.Cmd.Mode;
				robot->Cntrl.Int._Volts 		= robot->Cntrl.Cmd.Volts;
				robot->Cntrl.Int._Pinch 		= robot->Cntrl.Cmd.Pinch;

			break;

			case 21:

				if((robot->Cntrl.Cmd.Mode != robot->Cntrl.Int._Mode )
					|| (robot->Cntrl.Cmd.WFS != robot->Cntrl.Int._WFS)
					|| (robot->Cntrl.Cmd.Volts != robot->Cntrl.Int._Volts )
					|| (robot->Cntrl.Cmd.Pinch != robot->Cntrl.Int._Pinch )
					|| robot->Cntrl.Cmd.SendParam
					){

					robot->Cntrl.Cmd.SendParam = 0;

					robot->wc.setup.ctrlParam.ParameterMask = 0x0F; // 0b0001111; // change accordingly for Mode 5
					UINT *mode 	= &robot->Cntrl.Cmd.Mode; // Mode
					UINT WFS_SP = (UINT)(robot->Cntrl.Cmd.WFS * 1); //WF
					UINT VoltsSP = (UINT)(robot->Cntrl.Cmd.Volts * 10); //Volts
					UINT PinchSP = (UINT)(robot->Cntrl.Cmd.Pinch * 10); //Pinch

					if(robot->Cntrl.Cmd.Development)
						robot->wc.setup.ctrlParam.WeldMode = 0;
					else
						robot->wc.setup.ctrlParam.WeldMode = *mode;

					robot->wc.setup.ctrlParam.WorkPoint = WFS_SP;
					robot->wc.setup.ctrlParam.Trim = VoltsSP;
					robot->wc.setup.ctrlParam.WaveControl1 = PinchSP;

					// This command write Controls Parameter into Power Supply
					intrf->xCMD = ROBOT_SET_CONTROLS;

					robot->Cntrl.Int._Mode 			= robot->Cntrl.Cmd.Mode;
					robot->Cntrl.Int._WFS 			= robot->Cntrl.Cmd.WFS;
					robot->Cntrl.Int._Volts 		= robot->Cntrl.Cmd.Volts;
					robot->Cntrl.Int._Pinch 		= robot->Cntrl.Cmd.Pinch;

				}

			break;

			case 22:

				if((robot->Cntrl.Cmd.Mode != robot->Cntrl.Int._Mode )
					|| (robot->Cntrl.Cmd.WFS != robot->Cntrl.Int._WFS)
					|| (robot->Cntrl.Cmd.Trim != robot->Cntrl.Int._Trim )
					|| (robot->Cntrl.Cmd.UltimArc != robot->Cntrl.Int._UltimArc )
					|| robot->Cntrl.Cmd.SendParam
					){

					robot->Cntrl.Cmd.SendParam = 0;

					robot->wc.setup.ctrlParam.ParameterMask = 0x0F; // 0b0001111; // change accordingly for Mode 5
					UINT *mode 	= &robot->Cntrl.Cmd.Mode; // Mode
					UINT WFS_SP = (UINT)(robot->Cntrl.Cmd.WFS * 1); // WF
					UINT TrimSP = (UINT)(robot->Cntrl.Cmd.Trim * 100); // Trim
					UINT UltimArcSP = (UINT)(robot->Cntrl.Cmd.UltimArc * 10); //Pinch

					if(robot->Cntrl.Cmd.Development)
						robot->wc.setup.ctrlParam.WeldMode = 0;
					else
						robot->wc.setup.ctrlParam.WeldMode = *mode;

					robot->wc.setup.ctrlParam.WorkPoint = WFS_SP;
					robot->wc.setup.ctrlParam.Trim = TrimSP;
					robot->wc.setup.ctrlParam.WaveControl1 = UltimArcSP;

					// This command write Controls Parameter into Power Supply
					intrf->xCMD = ROBOT_SET_CONTROLS;

					robot->Cntrl.Int._Mode 			= robot->Cntrl.Cmd.Mode;
					robot->Cntrl.Int._WFS 			= robot->Cntrl.Cmd.WFS;
					robot->Cntrl.Int._Trim 			= robot->Cntrl.Cmd.Trim;
					robot->Cntrl.Int._UltimArc 		= robot->Cntrl.Cmd.UltimArc;

				}

			break;

			case 160:
			case 161:
			case 162:
			case 163:
			case 164:
			case 165:
			case 166:
			case 167:

				if((robot->Cntrl.Cmd.Mode != robot->Cntrl.Int._Mode )
					|| (robot->Cntrl.Cmd.Volts != robot->Cntrl.Int._Volts )
					//|| (robot->Cntrl.Cmd.Pinch != robot->Cntrl.Int._Pinch )
					){

					robot->wc.setup.ctrlParam.ParameterMask = 0x03; // 0b0000011; // Volts and WaveCntr 1

					//robot->wc.setup.ctrlParam.ParameterMask = 0x01; // Only Volts

					UINT *mode 	= &robot->Cntrl.Cmd.Mode; // Mode
					UINT VoltsSP = (UINT)(robot->Cntrl.Cmd.Volts * 10); // Volts
					robot->wc.setup.ctrlParam.WeldMode = *mode;
					robot->wc.setup.ctrlParam.WorkPoint = VoltsSP;
					//robot->wc.setup.ctrlParam.WaveControl1 = (UINT)(robot->Cntrl.Cmd.Pinch * 10);
					robot->wc.setup.ctrlParam.WaveControl1 = 0;

					// This command write Controls Parameter into Power Supply
					intrf->xCMD = ROBOT_SET_CONTROLS;

				}

				robot->Cntrl.Int._Mode 			= robot->Cntrl.Cmd.Mode;
				robot->Cntrl.Int._Volts 		= robot->Cntrl.Cmd.Volts;
				//robot->Cntrl.Int._Pinch 		= robot->Cntrl.Cmd.Pinch;

			break;

			case 170:

				if((robot->Cntrl.Cmd.Mode != robot->Cntrl.Int._Mode )
					|| (robot->Cntrl.Cmd.WFS != robot->Cntrl.Int._WFS)
					|| (robot->Cntrl.Cmd.Volts != robot->Cntrl.Int._Volts )
					|| (robot->Cntrl.Cmd.UltimArc != robot->Cntrl.Int._UltimArc )
					|| robot->Cntrl.Cmd.SendParam
					){

					robot->Cntrl.Cmd.SendParam = 0;

					robot->wc.setup.ctrlParam.ParameterMask = 0x0F; // 0b0001111; // change accordingly for Mode 5
					UINT *mode 	= &robot->Cntrl.Cmd.Mode; // Mode
					UINT WFS_SP = (UINT)(robot->Cntrl.Cmd.WFS * 1); //WF
					UINT VoltsSP = (UINT)(robot->Cntrl.Cmd.Volts * 10); //Volts
					UINT UltimArcSP = (UINT)(robot->Cntrl.Cmd.UltimArc * 10); //UltimArc

					if(robot->Cntrl.Cmd.Development)
						robot->wc.setup.ctrlParam.WeldMode = 0;
					else
						robot->wc.setup.ctrlParam.WeldMode = *mode;

					robot->wc.setup.ctrlParam.WorkPoint = WFS_SP;
					robot->wc.setup.ctrlParam.Trim = VoltsSP;
					robot->wc.setup.ctrlParam.WaveControl1 = UltimArcSP;

					// This command write Controls Parameter into Power Supply
					intrf->xCMD = ROBOT_SET_CONTROLS;

					robot->Cntrl.Int._Mode 			= robot->Cntrl.Cmd.Mode;
					robot->Cntrl.Int._WFS 			= robot->Cntrl.Cmd.WFS;
					robot->Cntrl.Int._Volts 		= robot->Cntrl.Cmd.Volts;
					robot->Cntrl.Int._UltimArc 		= robot->Cntrl.Cmd.UltimArc;

				}

			break;

			case 200:  // Calibration Current

				if((robot->Cntrl.Cmd.Mode != robot->Cntrl.Int._Mode )
					|| (robot->Cntrl.Cmd.AmpSP != robot->Cntrl.Int._AmpSP )
					){

					robot->wc.setup.ctrlParam.ParameterMask = 0x03; // 0b0000011; // change accordingly for Mode 200
					UINT *mode 	= &robot->Cntrl.Cmd.Mode; // Mode
					UINT AmpSP = (UINT)(robot->Cntrl.Cmd.AmpSP * 1); //amps
					robot->wc.setup.ctrlParam.WeldMode = *mode;
					robot->wc.setup.ctrlParam.WorkPoint = AmpSP;

					// This command write Controls Parameter into Power Supply
					intrf->xCMD = ROBOT_SET_CONTROLS;

				}

				robot->Cntrl.Int._Mode 			= robot->Cntrl.Cmd.Mode;
				robot->Cntrl.Int._AmpSP 		= robot->Cntrl.Cmd.AmpSP;

			break;

		}

	}
	//********************************************************//

	//*****************Lowest Priority CMD ********************//
	if(!intrf->xCMD){
		if(robot->Cntrl.Cmd.RST != robot->Cntrl.Int._RST){

			robot->Cntrl.Fbk.Status = 0;
			robot->miscSetup.state = 0; //reset misc state machine state
			robot->miscSetup.CoolerAddr = 0;
			robot->isMapping = 0;
			robot->isMapped = 0;	    //clear flag, set to unmapped status, stop timer
			robot->isMiscSetupOneShot = 0;
			robot->Comm.ArcComTimer.IN = 0;
			robot->Comm.StopRespondHeartBeat = 1; //halt heartbeat,force master to send out RESET request

		}
		robot->Cntrl.Int._RST 			= robot->Cntrl.Cmd.RST;

	}

	//*************** FEEDBACK  *****************************/

	robot->Cntrl.Fbk.curArcVolt = robot->wc.data.telemetry.fVoltage;
	robot->Cntrl.Fbk.curArcAmp  = robot->wc.data.telemetry.fCurrent;
	//robot->Cntrl.Fbk.Error      =  ???????
	//robot->Cntrl.Fbk.Status      =  ???????

	//********************************************************//

	return;

}

void error_status_handler(Arc_Link_typ *arc)
{

	Robot_typ *robot;
	if(!arc) return;

	robot = &arc->robot;

	// System is ready when mapped, ready status from PS is set and Arc Link Active, could add no system fault here
	if ((robot->isReady) && (robot->isMapped) && (robot->Comm.ArcLinkActive) && !robot->Cntrl.Fbk.Error)
	{
		robot->Cntrl.Fbk.Status |= PS_Ready;
//		log_event(&robot->eventlog , "Power supply is ready");
	}

	else
		robot->Cntrl.Fbk.Status &= ~PS_Ready;

	/*
	if ((robot->Cntrl.Fbk.Error >> 1 & 0x0001) || (robot->Cntrl.Fbk.Error >> 2 & 0x0001))  //either system fault from PS or network error will generate fault condition
		robot->Cntrl.Fbk.Error |= PS_Error_Present;
	else
		robot->Cntrl.Fbk.Error &= ~PS_Error_Present;
	*/
}
void ArcLink_Timer(Arc_Link_typ *arc){
//
	Robot_typ *robot;
	if(!arc) return;

	robot = &arc->robot;

	robot->Comm.PT = 2000; // 2s  timeout

	robot->Comm.CoolerSensPull_PT = 500; // 0.5s  timer

    robot->Comm.ArcComTimer.PT = robot->Comm.PT;

	if (robot->Comm.HeartBeat_Received && (robot->Comm.ArcComTimer.ET > 0)) //everytime got heartbeat, reset timer, to prevent trigger timeout
	    robot->Comm.ArcComTimer.IN = 0;

	else if (robot->Comm.HeartBeat_Received && (robot->Comm.ArcComTimer.ET == 0)){ //start timer, reset heartbeat flag
		if (robot->isMapped){  //
			robot->Comm.ArcComTimer.IN = 1;
		}
		if (robot->Comm.ClearError)    // clear error once getting connectivity from PS
		{
			robot->Comm.ClearError = 0;
			robot->Cntrl.Fbk.Error = 0;
			log_event(&robot->eventlog , "Network is active");
		}
		robot->Comm.HeartBeat_Received = 0;   //reset flag to start watchdog

	}

	TON(&robot->Comm.ArcComTimer);  //2 seconds Watchdog

    if (!robot->Comm.ArcComTimer.Q)
	robot->Comm.ArcLinkActive = 1;  // 1 Active
	else
	robot->Comm.ArcLinkActive = 0;	//timeout

	if (!robot->Comm.ArcLinkActive)
	{
		DBG_OB("Arc Link Disconnected\r\n");
		robot->Cntrl.Fbk.Error |= ArcLink_Com_Failed;
		robot->Cntrl.Fbk.Status = 0;
		robot->isMapping = 0;
		robot->isMapped = 0;	    //clear flag, set to unmapped status, stop timer
		robot->isMiscSetupOneShot = 0;
		robot->Comm.ArcComTimer.IN = 0;
		robot->Comm.ClearError = 1;	 //set flag when getting communication back, reset error
		log_event(&robot->eventlog , "Network is down");
	}
	else if (robot->isMapped)
	{
	/*	DBG_OB("Arc Link Connected\r\n"); */
		robot->Cntrl.Fbk.Error &= ~ArcLink_Com_Failed;
		robot->Cntrl.Fbk.Status |= ArcLink_Active;

	}

	// Pull Cooler Sens Status

	if((robot->miscSetup.CoolerAddr > 0)
		&& (robot->Comm.CoolerSensPull_PT > 0)){

		robot->Comm.CoolerSensPullTimer.PT = robot->Comm.CoolerSensPull_PT;

		if(robot->isMapped && robot->Comm.ArcLinkActive){

			if(!robot->Comm.CoolerSensPullTimer.IN){
				readAttribute_CoolerSens(arc);
				DBG("commanded Get Cooler Sens! \r\n" );
				robot->Comm.CoolerSensPullTimer.IN = 1;
				//TON(&robot->Comm.CoolerSensPullTimer);
			}
			else if(robot->Comm.CoolerSensPullTimer.Q){

				robot->Comm.CoolerSensPullTimer.IN = 0;
				//TON(&robot->Comm.CoolerSensPullTimer);

			}
			//else
				//TON(&robot->Comm.CoolerSensPullTimer);

		}

		TON(&robot->Comm.CoolerSensPullTimer);
	}

}
#endif /* _ROBOT_C */
```

### Program Logical/Libraries/bglibas

#### bgssm.c
```c
/********************************************************************
 * COPYRIGHT -- belgor
 ********************************************************************
 * Library: bglibas
 * File: bglibas.c
 * Author: admin
 * Created: March 07, 2012
 ********************************************************************
 * Implementation of library bglibas
 ********************************************************************/

#include <bur/plctypes.h>
#ifdef __cplusplus
	extern "C"
	{
#endif

	#include "bglibas.h"

#ifdef __cplusplus
	};
#endif

#include <string.h>

/* Init state machine. MUST be called once, before any other bgSSM function call. */
unsigned long bgSSMInit(struct bgSSM_typ* p, unsigned long pFunGetStateName, unsigned long pFunCyclicCallback)
{
	/*TODO: Add your code here*/
	memset(p, 0, sizeof(struct bgSSM_typ));

	p->pfunGetStateName = (UDINT)pFunGetStateName;
	p->pfunCyclicCallback = (UDINT)pFunCyclicCallback;
	p->stateInit = 1;
	return(0);
}
/* State machine cyclic operation. */
unsigned long bgSSMCyclic(struct bgSSM_typ* p)
{
	/*TODO: Add your code here*/
	int ii;

	//operate all timers
	for(ii=0; ii<BGSSM_TIMER_COUNT;ii++){
		bgTimerCyclic(&p->timer_x1ms[ii]);
	}
	bgTimerCyclic(&p->dlytimer_x1ms);

	//operate dlyCycle counter
	if(p->dlyCycles){
		p->dlyCycles--;
	}

	//call cyclic callback function if defined
	if(p->pfunCyclicCallback){
		void(*callback)(bgSSM_typ*) = ( void (*) (bgSSM_typ*) ) p->pfunCyclicCallback;
		(*callback)(p);
	}

	//clear single cycle flag every scan
	p->stateInit = 0;

	//check if state change requested
	if(p->state != p->stateNext){

		//if state change w. delay > wait for delay timer to expire or dlyCycles == 0
		if(!bgTimerIsTimeOut(&p->dlytimer_x1ms) || p->dlyCycles){
			return 1;
		}

		p->state = p->stateNext;
		//generate stateInit sigle scan flag
		p->stateInit = 1;

		//define state name if exteranl function for state names is defined
		if( p->pfunGetStateName ){
			char*(*getStateName)(UDINT) = ( char* (*) (UDINT) )p->pfunGetStateName;
			strcpy(p->stateText, (*getStateName)(p->state));
		}else{
			strcpy(p->stateText, "???");
		}
	}
	return(0);
}
/* Change to next state. */
unsigned long bgSSMStateNext(struct bgSSM_typ* p, unsigned long stateNext)
{
	/*TODO: Add your code here*/
	p->stateNext = stateNext;
	return(p->stateNext);
}

/* Change to next state w. timer delay. */
unsigned long bgSSMStateNextTimeDelay(struct bgSSM_typ* p, unsigned long stateNext, unsigned long delayTimeX1ms)
{
	/*TODO: Add your code here*/
	p->stateNext = stateNext;
	bgTimerStart(&p->dlytimer_x1ms, delayTimeX1ms);
	return(p->stateNext);
}

/* Change to next state w. cycles delay. */
unsigned long bgSSMStateNextCycleDelay(struct bgSSM_typ* p, unsigned long stateNext, unsigned long delayCycles)
{
	/*TODO: Add your code here*/
	p->stateNext = stateNext;
	p->dlyCycles = delayCycles;
	return(p->stateNext);
}
/* Check if first scan for the state. */
plcbit bgSSMIsStateInit(struct bgSSM_typ* p)
{
	/*TODO: Add your code here*/
	return(p->stateInit);
}
//EOF

/* Get current state */
unsigned long bgSSMGetState(struct bgSSM_typ* p)
{
	/*TODO: Add your code here*/
	return(p->state);
}

/* Get current state text*/
plcstring* bgSSMGetStateText(struct bgSSM_typ* p)
{
	/*TODO: Add your code here*/
	return(&p->stateText[0]);
}
```

- Library Logical/Libraries/sprintf2 (ANSIC) (no source held here)

### udpApp.var
```iecst
(********************************************************************
 * COPYRIGHT -- HP
 ********************************************************************
 * File: Global.var
 * Author: goran
 * Created: January 23, 2013
 ********************************************************************
 * Global variables of project YieldPlus
 ********************************************************************)
VAR
	gTxEvent : BOOL := FALSE;
	gTxRply : BOOL := FALSE;
	gJsontextTxRply : STRING[PAI_PVILIGHT_UDP_MSG_SIZE_MAX];
	gJsontextRx : STRING[PAI_PVILIGHT_UDP_MSG_SIZE_MAX];
	gJsontext : STRING[PAI_PVILIGHT_UDP_MSG_SIZE_MAX];
END_VAR
```

### cJSON.var
```iecst
(********************************************************************
 * COPYRIGHT -- HP
 ********************************************************************
 * Package: cJSON
 * File: cJSON.var
 * Author: goran
 * Created: June 19, 2013
 ********************************************************************
 * Variables of package cJSON
 ********************************************************************)
VAR
	gPaiPVILists : paiPVIListCollection_typ := (0);
	gHashValuesArray : ARRAY[0..19] OF UDINT;
	mHashCalcDone : UDINT;
	mHashCalcDlyTmr : TON;
END_VAR
```

### Program Logical/UDP/paiUDPService/udpclient

#### udpclient.c
```c
/********************************************************************
 * COPYRIGHT -- belgor
 ********************************************************************
 * Program: udpclient
 * File: udpclient.c
 * Author: goran
 * Created: January 23, 2013
 ********************************************************************
 * Implementation of program udpclient
 ********************************************************************/

#include <bur/plctypes.h>

#ifdef _DEFAULT_INCLUDES
	#include <AsDefault.h>
#endif

#include <../../../bglib/bgstring.c>
//#include <../../../bglib/bgTimer1ms.c>
//#include <string.h>

enum{
	udpCliZero = 0,
	udpCliInit,
	udpCliOpen,
	udpCliConnect,
	udpCliIdle,
	udpCliTxData,
	udpCliDisconnect,
	udpCliClose,
	udpCliError,
	udpCliLast
}STATEMACHINE;

static const char* udpCliStateName(int state)
{
static const char* stateNames[] = {
"Zero",
"Init",
"Open",
"Connect",
"Idle",
"TxData",
"Disconnect",
"Close",
"Error",
};

	if( state >= udpCliLast)
		return "unknow";

	return stateNames[state];
};

#define UDP_TX_BUF_SIZE_DEVICEDRIVER 100000
_LOCAL UDINT udpTxBufSize;

/*
###############################################################################
Utilities
###############################################################################
*/

static void convertIPTextToDigits(udpIPAddress_typ* p)
{
unsigned char txtbuffer[64];
bgStringList_typ list;

	strcpy((void*)txtbuffer, (void*)(p->text));
	list.src = txtbuffer;

	bgStringSplitLine(&list, '.');
	if(list.itemCount != 4){
		p->digit3 = 0;
		p->digit2 = 0;
		p->digit1 = 0;
		p->digit0 = 0;
		return;
	}
	p->digit3 = (USINT)atoi((UDINT)list.items[0]);
	p->digit2 = (USINT)atoi((UDINT)list.items[1]);
	p->digit1 = (USINT)atoi((UDINT)list.items[2]);
	p->digit0 = (USINT)atoi((UDINT)list.items[3]);
}

/**
 Simple logging
 Log goes to an array of PV strings > see _LOCAL STRING log[][] variable below
 Log output is visible via Automation Studio watch window
 Example of a log statement used within the code is:
 DBG(lgr, "This is log example. %d ", value1);
 To complety disable logging from this source file, change next line to: #if 0
*/
#if 1
#include <../../../bglib/bgPVLogger.c>
#define LOG_ENTRY_COUNT 20	//max number of log entries
#define LOG_ENTRY_LENGTH  32 //max length of individual log message. Longer msg are truncated
_LOCAL STRING log[LOG_ENTRY_COUNT][LOG_ENTRY_LENGTH]; //log output visible from Automation Studio!
static bgPVLogger_typ lgr;	//PV logger object
#else
#define DBG(loggerInstance, format, args...) ;
#define DBGINIT(loggerInstance, logoutput, logEntryCount, logEntrySize)  ;
#endif

/*
###############################################################################
Functions
###############################################################################
*/

static void udpClientSMCyclic(udpClient_typ *p)
{
bgSSM_typ* pSm = &p->sm;

	//operate timer(s)
	bgTimerCyclic(&pSm->timer_x1ms[0]); // delay timer

	//TimerExecute(&pSm->timer2x1ms); // update rate timer (in continues mode)
	//IMPORANT: for high speed, can't use TON block > rather, use cycle time
	if(pSm->timer_x1ms[1].ET)
		pSm->timer_x1ms[1].ET--;

	bgTimerCyclic(&pSm->timer_x1ms[2]); // 1sec stats timer

	//stats timers
	if( bgTimerIsTimeOut(&pSm->timer_x1ms[2]) ){
		bgTimerStart(&pSm->timer_x1ms[2], 1000);

		//values for cummulative (per min) calculations for datagrams
		p->txStats.datagramPerSec = pSm->counter[0];
		pSm->counter[0] = 0;
		if(p->txStats.datagramPerSec > p->txStats.datagramPerSecMax){
			p->txStats.datagramPerSecMax = p->txStats.datagramPerSec;
		}

		//values for cummulative (per min) calculations for bytes
		p->txStats.bytesPerSec = pSm->counter[1];
		pSm->counter[1] = 0;
		if(p->txStats.bytesPerSec > p->txStats.bytesPerSecMax){
			p->txStats.bytesPerSecMax = p->txStats.bytesPerSec;
		}
	}

	/*execute control state machine cyclic handler*/
	bgSSMCyclic(pSm);

	//show change of state in a log
	if( bgSSMIsStateInit(pSm) ){
		DBG(lgr, "sm=%s(%d)", bgSSMGetStateText(pSm), bgSSMGetState(pSm));
	}

	switch( bgSSMGetState(pSm) ){
		//========================================
		case udpCliZero:
			bgSSMStateNext(pSm, udpCliInit);
		break;
		//========================================
		case udpCliInit:
			if(p->clientIf.iConnect){
				bgSSMStateNext(pSm, udpCliOpen);
			}
		break;
		//========================================
		case udpCliOpen:

			if( bgSSMIsStateInit(pSm) ){
				p->client.open.enable = 1;
				p->client.open.port = 0;
				p->client.open.pIfAddr = 0;
//IMPORTANT:
//in order for the following conditional compilation to work properly, PLC object in the Configuration view
//must contain following defintion:
//Folder: Build
//Field: Additional Build Options
//Value: -D $(AS_CONFIGURATION)
//Using the above, name of the current AS configuration (i.e. realhw1 or testsim or else) becomes
//a defined preprocessor name. As a result, it's possible to destinguish between different configurations!
#ifdef Simulation
				//In case of testsim (ARsim) target, don't use socket options
				p->client.open.options = 0;
#warning "ISM Project - ARsim target!"
#else
				//For all other (real) targets, use socket options
				p->client.open.options = udpOPT_REUSEPORT | udpOPT_BROADCAST;
#warning "ISM Project - real target!"
#endif
				return;
			}

			if(p->client.open.status == ERR_FUB_BUSY)
				return;

			p->client.open.enable = 0;

			if(p->client.open.status == ERR_OK){
				p->client.recv.ident = p->client.open.ident;
				p->client.send.ident = p->client.open.ident;
				p->client.close.ident = p->client.open.ident;
				p->client.connect.ident = p->client.open.ident;
				p->client.disconnect.ident = p->client.open.ident;
				p->client.ioctl.ident = p->client.open.ident;

				udpTxBufSize = UDP_TX_BUF_SIZE_DEVICEDRIVER;
				p->client.ioctl.pData = &udpTxBufSize;
				p->client.ioctl.datalen = sizeof(udpTxBufSize);
				p->client.ioctl.ioctl = udpSO_SNDBUF_SET;
				p->client.ioctl.enable = 1;

				bgSSMStateNext(pSm, udpCliConnect);
				return;
			}

			DBG(lgr,"Err udp.open=%d", p->client.open.status);
			bgSSMStateNext(pSm, udpCliError);

		break;
		//========================================
		case udpCliConnect:

			if( bgSSMIsStateInit(pSm) ){
				p->client.connect.enable = 1;
				p->client.connect.port = p->clientIf.iRmtUdpPort;
				p->client.connect.pHost = (UDINT)p->clientIf.iRmtIPAddr;
				p->client.ioctl.enable = 0;
				return;
			}

			if(p->client.connect.status == ERR_FUB_BUSY)
				return;

			//p->client.connect.enable = 0;

			if(p->client.connect.status == ERR_OK){
				strcpy(p->clientIf.oRmtIpAddr, p->clientIf.iRmtIPAddr);
				p->clientIf.oRmtUdpPort = p->clientIf.iRmtUdpPort;

				bgSSMStateNext(pSm, udpCliIdle);
				return;
			}

			DBG(lgr,"Err udp.connect=%d", p->client.connect.status);
			bgSSMStateNext(pSm, udpCliError);

		break;
		//========================================
		case udpCliIdle:

			if( bgSSMIsStateInit(pSm) ){

			}

			if(!p->clientIf.iConnect){
				DBG(lgr,"disconnect request");
				bgSSMStateNext(pSm, udpCliDisconnect);
				return;
			}

			//udp client in echo mode!?
			//check for iSendEcho set by the server upon it receives a message > client sends out to the same host
			if((p->clientIf.iMode == 0) && p->clientIf.iSendEcho){
				p->clientIf.iSendEcho = 0;
				p->clientIf.iSend = 1;
				strcpy(p->clientIf.iRmtIPAddr, p->clientIf.iSendEchoRmtIpAddr);
			}

			//udp client in continues mode!?
			//trigger send update at a configured rate to a defined (sipplied to the inputs) remote host/port
			if(p->clientIf.iMode == 1){

				if(!pSm->timer_x1ms[1].ET){
					int updateTimeMs;

					if( p->clientIf.iUpdateRate ){
						updateTimeMs = 1000 /  p->clientIf.iUpdateRate;
					}else{
						updateTimeMs = 1000;
					}

					if(updateTimeMs < 10)
						updateTimeMs = 12;

					if(updateTimeMs > 1000)
						updateTimeMs = 1000;

					if(p->clientIf.iTaskCycleTimeXms){
						pSm->timer_x1ms[1].ET= updateTimeMs / p->clientIf.iTaskCycleTimeXms;
					}else{
						pSm->timer_x1ms[1].ET= updateTimeMs / gUdpClient_TaskCycleTimeXms; // devide by task clas time to find out increments
					}

					p->clientIf.iSend = 1;
				}
			}

			//monitor for change in remote host settings
			//in case of a change > reconnect (disconncet then connect)
			if((p->clientIf.oRmtUdpPort != p->clientIf.iRmtUdpPort) ||
				strcmp(p->clientIf.oRmtIpAddr, p->clientIf.iRmtIPAddr)
			){
				DBG(lgr,"rmt settings changed. Triggering reconnect.");
				bgSSMStateNext(pSm, udpCliDisconnect);
				return;
			}

			//monitor request to send
			if(!p->clientIf.iSend){
				return;
			}
			p->clientIf.iSend = 0;

			if(p->clientIf.iTxDataLen > UDP_CLIENT_TXBUF_SIZE){
				p->clientIf.iTxDataLen = UDP_CLIENT_TXBUF_SIZE;
			}

			if(!p->clientIf.iTxDataAdr && !p->clientIf.iTxCallback){
				DBG(lgr,"udp.send nothing to tx");
				return;
			}

			//execute memcpy if datasource is defined
			if(p->clientIf.iTxDataAdr){
				memcpy((void*)(p->txbuf), (void*)(p->clientIf.iTxDataAdr), p->clientIf.iTxDataLen);
			}

			//execute callback to enable app to populate data before sending
			//NOTE: callback will overwrite effect of the above memcpy if both a defined!!!
			if(p->clientIf.iTxCallback){
				void (*txCallback)(UDINT pBuf, UDINT lenTxBuf, UDINT* pLenData) =  ( void(*) (UDINT, UDINT, UDINT*) ) p->clientIf.iTxCallback;
				(*txCallback)( (UDINT)&p->txbuf[0], UDP_CLIENT_TXBUF_SIZE, &p->clientIf.iTxDataLen);
			}

			//don't trigger send if data len == 0
			if(!p->clientIf.iTxDataLen){
				bgSSMStateNext(pSm, udpCliIdle);
				return;
			}

			p->client.send.enable = 1;
			p->client.send.pData = (UDINT)&p->txbuf[0];
			p->client.send.datalen = p->clientIf.iTxDataLen;

			//stats
			p->txStats.datagramCountTotal++;
			p->txStats.bytesTotal += p->client.send.datalen;

			//values for cummulative (per min) calculations
			pSm->counter[0]++;
			pSm->counter[1] +=p->client.send.datalen;

			bgSSMStateNext(pSm, udpCliTxData);

		break;
		//========================================
		case udpCliTxData:
			if( bgSSMIsStateInit(pSm) ){

			}

			if(p->client.send.status == ERR_FUB_BUSY)
				return;

			p->client.send.enable = 0;

			if(p->client.send.status == ERR_OK){
				p->clientIf.oSendDone = 1;
				DBG(lgr,"udp.send OK");
				bgSSMStateNext(pSm, udpCliIdle);
				return;
			}

			DBG(lgr,"Err udp.send=%d", p->client.send.status);
			bgSSMStateNext(pSm, udpCliError);

		break;
		//========================================
		case udpCliDisconnect:

			if( bgSSMIsStateInit(pSm) ){
				p->client.connect.enable = 0;
				p->client.disconnect.enable = 1;
				return;
			}

			if(p->client.disconnect.status == ERR_FUB_BUSY)
				return;

			p->client.disconnect.enable = 0;

			if(p->client.disconnect.status == ERR_OK){
				bgSSMStateNext(pSm, udpCliClose);
				return;
			}

			DBG(lgr,"Err udp.disconnect=%d", p->client.disconnect.status);
			bgSSMStateNext(pSm, udpCliClose);

		break;
		//========================================
		case udpCliClose:

			if( bgSSMIsStateInit(pSm) ){
				DBG(lgr,"UDP Client close");
				p->client.close.enable = 1;
				return;
			}

			if(p->client.close.status == ERR_FUB_BUSY)
				return;

			if(p->client.close.status){
				DBG(lgr,"Err udp.close=%d", p->client.close.status);
			}

			p->client.close.enable = 0;

			bgSSMStateNext(pSm, udpCliZero);
		break;
		//========================================
		case udpCliError:

			if( bgSSMIsStateInit(pSm) ){
				DBG(lgr,"UDP Client Error State");

				//start error recovery timer
				bgTimerStart(&pSm->timer_x1ms[0], 5000);
			}

			if( bgTimerIsTimeOut(&pSm->timer_x1ms[0]) ){
				//after timer exp > try to close the port and see if it recovers
				bgSSMStateNext(pSm, udpCliDisconnect);
			}

		break;
		//========================================
		default:
		break;
	}

}

static void udpClientInit(udpClient_typ *p)
{
	bgSSM_typ* pSm = &p->sm;

	bgTimerStart(&p->sm.timer_x1ms[2], 1000);

	bgSSMInit(pSm, (UDINT)udpCliStateName, 0);

}

static void udpClientCyclic(udpClient_typ *p)
{

	//udp client state machine
	udpClientSMCyclic(p);

	//udp client fbk-s
	UdpOpen(&p->client.open);
	UdpClose(&p->client.close);
	UdpConnect(&p->client.connect);
	UdpDisconnect(&p->client.disconnect);
	UdpSend(&p->client.send);
	UdpRecv(&p->client.recv);
	UdpIoctl(&p->client.ioctl);
}

/*
###############################################################################
Main entry: Init & Cyclic Functions
###############################################################################
*/

void _INIT udpclientINIT(void)
{
	/* TODO: Add code here */

	//init logger object
	DBGINIT(lgr, log, LOG_ENTRY_COUNT, LOG_ENTRY_LENGTH);

	udpClientInit(&gUdpClient);

	//upd client application specific init
	//gUdpClient.clientIf.iConnect = 1;

	//RESTORE SETTINGS FROM THE REMANENT STORAGE
	//sanity check for remote host ip address
	convertIPTextToDigits(&gUdpSystemCfg.udpRemoteHostIpAddress);

	if(!gUdpSystemCfg.udpRemoteHostIpAddress.digit0 ||
		!gUdpSystemCfg.udpRemoteHostIpAddress.digit1 ||
		!gUdpSystemCfg.udpRemoteHostIpAddress.digit2 ||
		!gUdpSystemCfg.udpRemoteHostIpAddress.digit3
	){
		strcpy(gUdpSystemCfg.udpRemoteHostIpAddress.text, gUdpClient_DefaultHostAdr);
		convertIPTextToDigits(&gUdpSystemCfg.udpRemoteHostIpAddress);
	}
	strcpy(gUdpClient.clientIf.iRmtIPAddr, gUdpSystemCfg.udpRemoteHostIpAddress.text);

	//sanity check for remote host UDP port number
	if(!gUdpSystemCfg.udpRemoteHostPortNumber){
		gUdpSystemCfg.udpRemoteHostPortNumber = gUdpClient_DefaultPort;
	}
	gUdpClient.clientIf.iRmtUdpPort = gUdpSystemCfg.udpRemoteHostPortNumber;

	// udpClientMode
	// 0-echo mode (send status after receiving a command from the host. Uses received IP address and UDP port number configured here.
	// 1-continues mode (send status independantly to configured 	remoteIpAddress. remoteUDP port at the configure UDP rate
	// 2-user mode (send controled by the application via udp client IF)
	if(gUdpSystemCfg.udpClientMode > 2){
		gUdpSystemCfg.udpClientMode = 2;
	}
	gUdpClient.clientIf.iMode = gUdpSystemCfg.udpClientMode;

	// udpClientUpdateRate
	// rate to send outgoing status to remote host in case of UDP client mode 1
	//
	if(gUdpSystemCfg.udpClientUpdateRate < 1){
		gUdpSystemCfg.udpClientUpdateRate  = 1;
	}
	if(gUdpSystemCfg.udpClientUpdateRate > 100){
		gUdpSystemCfg.udpClientUpdateRate  = 100;
	}
	gUdpClient.clientIf.iUpdateRate = gUdpSystemCfg.udpClientUpdateRate;

	gUdpClient.clientIf.iSend = 0;

}

void _CYCLIC udpclientCYCLIC(void)
{
	/* TODO: Add code here */

	//udp client cyclic
	udpClientCyclic(&gUdpClient);

	//in continues client mode, use localy configured settings!
	if((gUdpSystemCfg.udpClientMode == 1) &&
		((gUdpSystemCfg.udpClientMode != gUdpClient.clientIf.iMode) ||
		(gUdpClient.clientIf.iUpdateRate != gUdpSystemCfg.udpClientUpdateRate) ||
		strcmp(gUdpClient.clientIf.iRmtIPAddr, gUdpSystemCfg.udpRemoteHostIpAddress.text))
	){
		gUdpClient.clientIf.iMode = gUdpSystemCfg.udpClientMode;
		gUdpClient.clientIf.iUpdateRate = gUdpSystemCfg.udpClientUpdateRate;
 		strcpy(gUdpClient.clientIf.iRmtIPAddr, gUdpSystemCfg.udpRemoteHostIpAddress.text);
		//use configured port number for the remote UDP host
		gUdpClient.clientIf.iRmtUdpPort = gUdpSystemCfg.udpRemoteHostPortNumber;
	}

	//in echo mode, just monitor for iMode change
	if((gUdpSystemCfg.udpClientMode == 0) &&
		((gUdpSystemCfg.udpClientMode != gUdpClient.clientIf.iMode) )
	){
		gUdpClient.clientIf.iMode = gUdpSystemCfg.udpClientMode;
		//use configured port number for the remote UDP host
		gUdpClient.clientIf.iRmtUdpPort = gUdpSystemCfg.udpRemoteHostPortNumber;
	}

	//in user mode, nothing todo
	if((gUdpSystemCfg.udpClientMode == 2) &&
		((gUdpSystemCfg.udpClientMode != gUdpClient.clientIf.iMode) )
	){
		gUdpClient.clientIf.iMode = gUdpSystemCfg.udpClientMode;
	}

}
```

### Program Logical/UDP/udpApp

#### udpApp.c
```c
/********************************************************************
 * COPYRIGHT -- belgor
 ********************************************************************
 * Program: appUDP
 * File: appUDP.c
 * Author: goran
 * Created: Jan 25, 2013
 ********************************************************************
 * Implementation of program appUDP
 ********************************************************************/

#include <bur/plctypes.h>

#ifdef _DEFAULT_INCLUDES
	#include <AsDefault.h>
#endif
//#include <string.h>

#include <../../bglib/bgString.c>
#include <../../bglib/bgBitUtilities.c>

/*
###############################################################################
Utilities
###############################################################################
*/

/**
 Simple logging
 Log goes to an array of PV strings > see _LOCAL STRING log[][] variable below
 Log output is visible via Automation Studio watch window
 Example of a log statement used within the code is:
 DBG(lgr, "This is log example. %d ", value1);
 To complety disable logging from this source file, change next line to: #if 0
IMPORTANT:
==========
DBGINIT() statement MUST BE PLACED as a first statement within the task _INIT function!
Example:
void _INIT myTaskINIT(void)
{
	//TODO: Add code here
	//init logger object
	DBGINIT(lgr, log, LOG_ENTRY_COUNT, LOG_ENTRY_LENGTH);
}
*/
#if 1
#include <../../bglib/bgPVLogger.c>
#define LOG_ENTRY_COUNT 20	//max number of log entries
#define LOG_ENTRY_LENGTH  32 //max length of individual log message. Longer msg are truncated
_LOCAL STRING log[LOG_ENTRY_COUNT][LOG_ENTRY_LENGTH]; //log output visible from Automation Studio!
static bgPVLogger_typ lgr;	//PV logger object
#else
#define DBG(loggerInstance, format, args...) ;
#define DBGINIT(loggerInstance, logoutput, logEntryCount, logEntrySize)  ;
#endif

//UDP Server Receive function
static void udpServerCallback(UDINT pRxBuffer, UDINT lenRxData)
{
	DBG(lgr, "udp rx, datalen=%d", lenRxData);
	if(lenRxData > sizeof(gJsontextRx)){
		DBG(lgr, "udp rx datalen(%d) TOO LONG!", lenRxData);
		return;
	}
	memcpy(gJsontextRx, pRxBuffer, lenRxData);
}

//UDP Server Receive function
static void udpServerCallbackAfterReceive(UDINT pRxBuffer, UDINT lenRxData)
{
	udpServerCallback(pRxBuffer, lenRxData);
}

//UDP Client Send Callback function
static void udpClientCallback(UDINT pTxBuffer, UDINT lenTxBuffer, UDINT* pTxDataLen)
{
int length;

	if(gTxRply){
		gTxRply = 0;
		strcpy( pTxBuffer, gJsontextTxRply );

		length = strlen(gJsontextTxRply);
		DBG(lgr, "udpClientCallback len1=%d", length);

		//define a total lenght of the message
		length = strlen(pTxBuffer);
		DBG(lgr, "udpClientCallback len2=%d", length);

		(*pTxDataLen) = length;

		DBG(lgr, "udpClientCallback[,20]: %s", &(((char*)pTxBuffer)[length -  20]));

		return;
	}else
	if(gTxEvent){
		gTxEvent = 0;
		strcpy( pTxBuffer, gJsontext );
		//define a total lenght of the message

		(*pTxDataLen) = strlen(pTxBuffer);

		DBG(lgr, "udp server rx timeout");

		return;
	}

	(*pTxDataLen) = 0;
}

//UDP Client Send Callback function
static void udpClientCallbackBeforeSend(UDINT pTxBuffer, UDINT lenTxBuffer, UDINT* pTxDataLen)
{
	udpClientCallback(pTxBuffer, lenTxBuffer, pTxDataLen);
}

static void	udpTimeOutHandler()
{
	//application logic - an example of handling a UDP receive timeout event
	static BOOL oldRxTimeout;
	if( gUdpServer.serverIf.oRxIsTimeout && !oldRxTimeout){
		DBG(lgr, "udp server rx timeout");
	}

	if( !gUdpServer.serverIf.oRxIsTimeout && oldRxTimeout){
		DBG(lgr, "udp server rx ok");
	}

	oldRxTimeout = gUdpServer.serverIf.oRxIsTimeout;
}

/*
###############################################################################
Task execution entry points: Init & Cyclic Functions
###############################################################################
*/
void _INIT udpAppINIT(void)
{
	/* TODO: Add code here */
	//init logger object
	DBGINIT(lgr, log, LOG_ENTRY_COUNT, LOG_ENTRY_LENGTH);

	//Define application specific UDP client tx callback function
	gUdpClient.clientIf.iTxCallback = (UDINT)udpClientCallbackBeforeSend;

	//Define application specific UDP server rx callback function
	gUdpServer.serverIf.iRxCallback = (UDINT)udpServerCallbackAfterReceive;
	gUdpServer.serverIf.oRxDataLenMax = (UDINT)sizeof(ctrlInterfaceCmd_typ);

	//Adjust UDP client/server settings according to the application needs (i.e. use HMI if needed)
	//For other defaults see:
	//paiUDPService.var (i.e. defined UDP related const)
	//udpserv.c/udpservINIT() and udpclient.c/udpclientINIT()
	gUdpSystemCfg.udpClientMode = 2;//user mode
	gUdpSystemCfg.udpClientUpdateRate = 20;//[Hz]
	//strcpy(gUdpSystemCfg.udpRemoteHostIpAddress.text, "192.168.100.31");
	//strcpy(gUdpSystemCfg.udpRemoteHostIpAddress.text, "192.168.100.171");
	strcpy(gUdpSystemCfg.udpRemoteHostIpAddress.text, "192.168.100.255");
	gUdpClient.clientIf.iTaskCycleTimeXms = 10;//udp client runs under 10ms cycle time
	gUdpServer.serverIf.iRxTimeoutXms = 4000;//udp server rx timeout time

}

void _CYCLIC udpAppCYCLIC(void)
{
	/* TODO: Add code here */

#if 0
	//application logic - on send complete, copy status into last statusSent
	if(gUdpClient.clientIf.oSendDone){
		gUdpClient.clientIf.oSendDone = 0;
		//save last transmitted data

	}

	//application logic - en example of handling a UDP rx event
	if(gUdpServer.serverIf.oRxReady){
		gUdpServer.serverIf.oRxReady = 0;

	}
#endif

	//handle a UDP rx timeout
	udpTimeOutHandler();
}
//EOF
```

### Program Logical/Universal/GasCoolPrc

#### GasCool.c
```c
/********************************************************************
 * COPYRIGHT -- wsi
 ********************************************************************
 * Program: GasCool
 * File: GasCool.c
 * Author: ckaczkowski
 * Created: March 05, 2014
 ********************************************************************
 * Implementation of program GasCool
 ********************************************************************/

#include <bur/plctypes.h>

#ifdef _DEFAULT_INCLUDES
	#include <AsDefault.h>
#endif

#include <..\..\Universal\SuperDeclaration.h>
#include <..\..\Lib\Statelib.c>
#include <..\..\Lib\WSI_lib.c>

_LOCAL TON_typ Tmr[GAS_NUM];
GenProcess_typ *prc;
GenProcess_typ *prcCool;

_LOCAL TON_typ CoolTmr[COOL_NUM];

_LOCAL  plcbit GasSolOutput[GAS_NUM];
_LOCAL  plcbit GasSwInput[GAS_NUM];
_LOCAL  plcbit CoolSolOutput[COOL_NUM];
_LOCAL  plcbit CoolSwInput[COOL_NUM];

_LOCAL TON_typ CoolTmo[COOL_NUM];
_LOCAL TON_typ GasTmo[GAS_NUM];

_LOCAL plcbit _GasTmoTrig[GAS_NUM] , _CoolTmoTrig[COOL_NUM];

_LOCAL plcbit Gas_Arclink_ON;
_LOCAL USINT ArcLink_Gas_Valve_step;

plcbit _gas_Arclink_ON;

void ArcLinkGasSol();

void _INIT GasCoolINIT(void)
{
	Process[0].Disable = Process[0].Disable;
}

void _CYCLIC GasCoolCYCLIC(void){
int i;

	//if(GAS_Param_Set[0].Mode == 1)
		ArcLinkGasSol();

	for(i=0 ; i < GAS_NUM ; i++){

			prc = GAS_Param_Set[i].pPrc;

			if(!prc)
				break;

			if(prc->ConfigReady <= 0)
				break;

			if(GAS_Param_Set[i].pSensInput)
				GasSwInput[i] = (*GAS_Param_Set[i].pSensInput);
			else
				GasSwInput[i] = GasSolOutput[i];

			if(prc->Disable){

				prc->_step = 0xFF;
				GasSolOutput[i]= 0;

				switch(prc->xCMD){

				case prcsForceON:
				case prcsSTART:

					prc->Status = prcsSTATUS_Run;

				break;

				case prcsHalt:
				case prcsRESTART:
				case prcsSTOP:

					prc->Status = prcsSTATUS_Stopped;

				break;

				default:

					if(!((prc->Status == prcsSTATUS_Stopped) || (prc->Status == prcsSTATUS_Run)))
						prc->Status = prcsSTATUS_Stopped;

				break;

				}

			}else{

				///////////////////////////////////
				switch(prc->xCMD){

					case prcsHalt:
					case prcsRESTART:

						prc->_step = 0;

					break;

					case prcsSTART:

					if((prc->_step) == 0 || (prc->_step > 5))
						prc->_step = 1;

					break;

					case prcsSTOP:

						if((prc->_step != 0) && (prc->_step <= 5))
							prc->_step = 20;

					break;

					case prcsForceON:

						prc->_step = 5;

					break;

				}
			}
			prc->xCMD = 0;

			/////////////////////////////////////

			switch(prc->_step){

				case 0:  // IDLE - stopped

					GasSolOutput[i]= 0;
					prc->Status = prcsSTATUS_Stopped;

				break;

				case 1: // start

					prc->Status = prcsSTATUS_StartDly;

					GasSolOutput[i]= 1;

					if(*GAS_Param_Set[i].pStartDly > 0.0){
						TimerStart(&Tmr[i],  *GAS_Param_Set[i].pStartDly);
						prc->_step = 2;
					}
					else
						prc->_step = 5;

				break;

				case 2:

					GasSolOutput[i]= 1;

					if(TimerIsTimeOut(&Tmr[i])){
						prc->_step = 5;

					}

				break;

				case 5:

					GasSolOutput[i]= 1;

					prc->Status = prcsSTATUS_Run;

				break;

				case 20:  // stop

					GasSolOutput[i]= 1;

					prc->Status = prcsSTATUS_StopDly;

					if(*GAS_Param_Set[i].pStopDly > 0){
						TimerStart(&Tmr[i], *GAS_Param_Set[i].pStopDly);
						prc->_step = 21;
					}
					else
						prc->_step = 0;

				break;

				case 21:

					GasSolOutput[i]= 1;

					if(TimerIsTimeOut(&Tmr[i]))
						prc->_step = 0;

				break;

			}

			TimerExecute(&Tmr[i]);

			if(TimerIsTimeOut(&GasTmo[i])){

				GasTmo[i].IN = 0;
				GasTmo[i].Q = 0;

				if(GasTmo[i].PT > 0){
					Errors(&ErrorMgr,ERROR_COOL_GAS ,ERROR_GAS_TMO,i);
					prc->_step = 0;
				}

			}
			else if(((!GasSwInput[i])&& GasSolOutput[i])
				&& !_GasTmoTrig[i]){

				TimerStart(&GasTmo[i],*GAS_Param_Set[i].pTmo);
				_GasTmoTrig[i] = 1;
			}

			else if(GasSwInput[i] || (!GasSolOutput[i])){

				GasTmo[i].IN = 0;
				GasTmo[i].Q = 0;

				_GasTmoTrig[i] = 0;

			}

		TimerExecute(&GasTmo[i]);
		if(GAS_Param_Set[i].pOutput)
			(*GAS_Param_Set[i].pOutput) = GasSolOutput[i];

	}

	///////////////////////////////////
	//  COOLANT
	//////////////////////////////////

	for(i=0 ; i < COOL_NUM ; i++){

			if(COOL_Param_Set[i].pSensInput)
				CoolSwInput[i] = (*COOL_Param_Set[i].pSensInput);
			else
				CoolSwInput[i] = CoolSolOutput[i];

			prcCool = COOL_Param_Set[i].pPrc;

			if(!prcCool)
				break;

			if(prcCool->ConfigReady <= 0)
				break;

			if(prcCool->Disable){

				prcCool->_step = 0xFF;
				CoolSolOutput[i]= 0;

				switch(prcCool->xCMD){

					case prcsSTART:

						prcCool->Status = prcsSTATUS_Run;

					break;

					case prcsHalt:
					case prcsSTOP:

						prcCool->Status = prcsSTATUS_Stopped;

					break;

					default:

						if(!((prcCool->Status == prcsSTATUS_Stopped) || (prcCool->Status == prcsSTATUS_Run)))
							prcCool->Status = prcsSTATUS_Stopped;

					break;

				}

			}
			else{

				///////////////////////////////////
				switch(prcCool->xCMD){

					case prcsHalt:
					case prcsSTOP:
					case prcsRESTART:

						CoolSolOutput[i]= 0;
						prcCool->Status = prcsSTATUS_Stopped;

					break;

					case prcsForceON:
					case prcsSTART:

						CoolSolOutput[i]= 1;
						prcCool->Status = prcsSTATUS_Run;

					break;

				}
			}

		prcCool->xCMD = 0;

		if(TimerIsTimeOut(&CoolTmo[i])){

			CoolTmo[i].IN = 0;
			CoolTmo[i].Q = 0;

			if(CoolTmo[i].PT > 0){
				Errors(&ErrorMgr,ERROR_COOL_GAS,ERROR_COOL_TMO,0);
				prcCool->xCMD = prcsHalt;
			}

		}

		else if(((!CoolSwInput[i])&& CoolSolOutput[i])
			&& !_CoolTmoTrig[i]){

			TimerStart(&CoolTmo[i],*COOL_Param_Set[i].pTmo);
			_CoolTmoTrig[i] = 1;
		}

		else if(CoolSwInput[i] || (!CoolSolOutput[i])){

			CoolTmo[i].IN = 0;
			CoolTmo[i].Q = 0;

			_CoolTmoTrig[i] = 0;

		}

		TimerExecute(&CoolTmr[i]);
		TimerExecute(&CoolTmo[i]);

		if(COOL_Param_Set[i].pOutput)
			(*COOL_Param_Set[i].pOutput) = CoolSolOutput[i];

	}
}
void ArcLinkGasSol(){
	/////////  GAS Solenoid ////

	Gas_Arclink_ON = GasSolOutput[0];

	if(!ArcLink.robot.isMapped){

		ArcLink_Gas_Valve_step = 2;

	}else{

		switch(ArcLink_Gas_Valve_step){

			default:

			break;

			case 1:

				if(ArcLink.robot.isMapped && (ArcLink.robot.miscSetup.state == 9)
					&& ArcLink.robot.isReady){

					if(!ArcLink.robot.Intrf.xCMD){

						ArcLink.robot.miscSetup.GasSolAddr = 0;
						ArcLink.robot.Intrf.xCMD = ROBOT_CMD_SEARCH_GAS_SOL_ADR;
						ArcLink_Gas_Valve_step ++;
					}

				}

			break;

			case 2:

				if(!ArcLink.robot.Intrf.xCMD
					&& (ArcLink.robot.miscSetup.GasSolAddr > 0)){

					_gas_Arclink_ON = !Gas_Arclink_ON;
					ArcLink_Gas_Valve_step ++;

				}

			break;

			case 3:

				if(!ArcLink.robot.Intrf.xCMD){

					if(Gas_Arclink_ON !=_gas_Arclink_ON){

						ArcLink.robot.Intrf.xCMD = ROBOT_CMD_GAS_SOL_ENABLE;
						ArcLink_Gas_Valve_step ++;

					}
				}

			break;

			case 4:

				if(!ArcLink.robot.Intrf.xCMD){

					if(Gas_Arclink_ON)
						ArcLink.robot.Intrf.xCMD = ROBOT_CMD_GAS_SOL_ON;

					else
						ArcLink.robot.Intrf.xCMD = ROBOT_CMD_GAS_SOL_OFF;

					ArcLink_Gas_Valve_step ++;

				}

			break;

			case 5:

				if(!ArcLink.robot.Intrf.xCMD){

					_gas_Arclink_ON = Gas_Arclink_ON;
					ArcLink_Gas_Valve_step = 3;

				}

			break;

		}

	}
	/////////////////////

}
```

### Program Logical/Universal/HW_PSprc

#### HW_PS.c
```c
/********************************************************************
 * COPYRIGHT -- wsi
 ********************************************************************
 * Program: HW_PS
 * File: HW_PS.c
 * Author: ckaczkowski
 * Created: November 26, 2013
 ********************************************************************
 * Implementation of program HW_PS
 ********************************************************************/

#include <bur/plctypes.h>

#ifdef _DEFAULT_INCLUDES
	#include <AsDefault.h>
#endif

#include <..\..\Universal\SuperDeclaration.h>
#include <..\..\Lib\Statelib.c>
#include <..\..\Lib\WSI_lib.c>

_LOCAL TON_typ Tmr[HW_PS_NUM];
GenProcess_typ* prc;
_LOCAL AzzRamp_typ Ramp[HW_PS_NUM];
_LOCAL  AzzLimScal_typ  LimScal_AmpCMD[HW_PS_NUM];

float _AmpSP[HW_PS_NUM];

void _INIT HW_PSINIT(void)
{
int i;

	Process[0].Disable = Process[0].Disable;
	Hardware[0].Anal_Inp[0] = Hardware[0].Anal_Inp[0];

	for(i=0 ; i < (HW_PS_NUM); i++){

		Ramp[i].y_max = 1000.0;
		Ramp[i].y_min = 0;
		Ramp[i].enable = 1;

		LimScal_AmpCMD[i].x1 = 0.0;
		LimScal_AmpCMD[i].y1 = 0.0;

	}

}

void _CYCLIC HW_PSCYCLIC(void)
{	int i;
	float y;

		for(i=0 ; i < HW_PS_NUM ; i++){

			prc = HW_PS_Param_Set[i].pPrc;

			if(!prc)
				break;

			if(!HW_PS_Param_Set[i].pCalibPoints)
				break;

			if(prc->ConfigReady <= 0)
				break;

			LimScal_AmpCMD[i].x2 = HW_PS_Param_Set[i].AmpCMD_Max;
			LimScal_AmpCMD[i].y2 = HW_PS_Param_Set[i].rawCmdMax;

			if(prc->Disable){

				prc->_step = 0xFF;

				switch(prc->xCMD){

					case prcsSTART:

						prc->Status = prcsSTATUS_Run;

					break;

					case prcsRESTART:
					case prcsHalt:
					case prcsSTOP:
					case prcsQuickSTOP:

						prc->Status = prcsSTATUS_Stopped;

					break;

					default:

						if(!((prc->Status == prcsSTATUS_Stopped) || (prc->Status == prcsSTATUS_Run)))
							prc->Status = prcsSTATUS_Stopped;

					break;

				}

			}else{

				///////////////////////////////////
				switch(prc->xCMD){

					case prcsRESTART:
					case prcsHalt:

						prc->_step = 0;

					break;

					case prcsForceON:

						if(prc->_step != 50)
							prc->_step = 50;

					break;

					case prcsJump2Run:

						if(prc->_step != 60)
							prc->_step = 60;

					break;

					case prcsCalib:

						if(prc->_step != 70)
							prc->_step = 70;

					break;

					case prcsSTART:

					if((prc->_step) == 0 || (prc->_step > 5))
						prc->_step = 1;

					break;

					case prcsQuickSTOP:
					case prcsSTOP:

						if((prc->_step != 0) && (prc->_step <= 5)){

							switch(prc->xCMD){

								case prcsQuickSTOP:

									prc->_step = 22;

								break;

								case prcsSTOP:

									prc->_step = 20;

								break;

							}

						}

					break;

					//test
					case 100:

					break;

				}
			}
			prc->xCMD = 0;

			/////////////////////////////////////

			switch(prc->_step){

				case 255: // Disable
				case 0:  // IDLE - stopped

					prc->Status = prcsSTATUS_Stopped;
					Ramp[i].y_set = 0.0;
					Ramp[i].set = 1;

				break;

				case 1: // start

					prc->Status = prcsSTATUS_StartDly;

					Ramp[i].y_set = *HW_PS_Param_Set[i].pStartAmp;
					Ramp[i].set = 1;

					if(*HW_PS_Param_Set[i].pStartDly > 0){
						TimerStart(&Tmr[i],  *HW_PS_Param_Set[i].pStartDly);
						prc->_step = 2;
					}
					else
						prc->_step = 3;

				break;

				case 2:

					Ramp[i].set = 1;

					if(TimerIsTimeOut(&Tmr[i])){
						prc->_step = 3;

					}

				break;

				case 3:

					prc->Status = prcsSTATUS_RampUp;

					if (*HW_PS_Param_Set[i].pRampUp > 0)
						Ramp[i].dy_up = fabsf((*HW_PS_Param_Set[i].pAmpSP - Ramp[i].y)/(*HW_PS_Param_Set[i].pRampUp));
					else
						Ramp[i].dy_up = 3.4e+38;

					Ramp[i].dy_down = Ramp[i].dy_up;
					Ramp[i].x = *HW_PS_Param_Set[i].pAmpSP;

					TimerStart(&Tmr[i],  *HW_PS_Param_Set[i].pRampUp);

					Ramp[i].set = 0;

					prc->_step = 4;

				break;

				case 4:

					if(Ramp[i].x_reached || TimerIsTimeOut(&Tmr[i])){
						_AmpSP[i] = (*HW_PS_Param_Set[i].pAmpSP);
						prc->_step = 5;

					}

				break;

				case 5:

					prc->Status = prcsSTATUS_Run;

					if(_AmpSP[i] != (*HW_PS_Param_Set[i].pAmpSP)){
						_AmpSP[i] = (*HW_PS_Param_Set[i].pAmpSP);

						Ramp[i].x = *HW_PS_Param_Set[i].pAmpSP;

						if (*HW_PS_Param_Set[i].pRampUp > 0)
							Ramp[i].dy_up = fabsf((*HW_PS_Param_Set[i].pAmpSP)/(*HW_PS_Param_Set[i].pRampUp));
							//Ramp[i].dy_up = fabsf((*HW_PS_Param_Set[i].pSpeedSp - Ramp[i].y)/(*HW_PS_Param_Set[i].pRampUp));
						else
							Ramp[i].dy_up = 3.4e+38;

						Ramp[i].dy_down = Ramp[i].dy_up;
					}

				break;

				case 20:

					prc->Status = prcsSTATUS_StopDly;

					if(*HW_PS_Param_Set[i].pStopDly > 0){
						TimerStart(&Tmr[i], *HW_PS_Param_Set[i].pStopDly);
						prc->_step ++;
					}
					else
						prc->_step = 22;

				break;

				case 21:

					if(TimerIsTimeOut(&Tmr[i]))
						prc->_step++;

				break;

				case 22:

					prc->Status = prcsSTATUS_RampDwn;

					if (*HW_PS_Param_Set[i].pRampDwn > 0)
						Ramp[i].dy_down = fabsf((Ramp[i].y - (*HW_PS_Param_Set[i].pEndAmp))/(*HW_PS_Param_Set[i].pRampDwn));
					else
						Ramp[i].dy_down = 3.4e+38;

					Ramp[i].dy_up = Ramp[i].dy_down;

					Ramp[i].x = *HW_PS_Param_Set[i].pEndAmp;

					TimerStart(&Tmr[i],  *HW_PS_Param_Set[i].pRampDwn);

					prc->_step++;

				break;

				case 23:

					if(Ramp[i].x_reached || TimerIsTimeOut(&Tmr[i]))
						prc->_step = 0;

				break;

				case 50:

					Ramp[i].y_set = *HW_PS_Param_Set[i].pStartAmp;
					Ramp[i].set = 1;

					prc->Status = prcsSTATUS_ForceON;

				break;

				case 60:

					_AmpSP[i] = (*HW_PS_Param_Set[i].pAmpSP);
					Ramp[i].y_set = _AmpSP[i];
					Ramp[i].x = _AmpSP[i];
					Ramp[i].set = 1;
					AzzRamp(&Ramp[i]);
					Ramp[i].set = 0;

					prc->_step = 5;

				break;

				case 70:

					prc->Status = prcsSTATUS_ForceCalib;

				break;

			}

			TimerExecute(&Tmr[i]);

			if(Ramp[i].dy_up <= 0.0){
				Ramp[i].dy_up = 3.4e+38;
				Ramp[i].dy_down = Ramp[i].dy_up;

			}
			AzzRamp(&Ramp[i]);

			if(HW_PS_Param_Set[i].pAnal_Output && HW_PS_Param_Set[i].pCalibPoints){

				prc->Fbk[1] = Ramp[i].y; // Cmd Amp

				if(prc->_step == 70){ // Calib

				   y = prc->fParam[1];

				   prc->Fbk[1] = 0; // Cmd Amp

				}
				else if(prc->Param[0])
					y = getFromCalib(Ramp[i].y, HW_PS_Param_Set[i].pCalibPoints , CALIB_2POINTS) ;

				else
					y = getFromCalib(Ramp[i].y, HW_PS_Param_Set[i].pCalibPoints , CALIB_2POINTS)  * ((*HW_PS_Param_Set[i].pAmpBoost)+1.0);

				(*HW_PS_Param_Set[i].pAnal_Output) = (INT)(LimScal( y , &LimScal_AmpCMD[i]));

			}

			if(	HW_PS_Param_Set[i].pOutput){

				if(prc->Status == prcsSTATUS_Stopped)

					(*HW_PS_Param_Set[i].pOutput) = 0;

				else
					(*HW_PS_Param_Set[i].pOutput) = ((*HW_PS_Param_Set[i].pAnal_Output)> 0);

			}

			if(!(HW_PS_Param_Set[i].pOutput))
				prc->Fbk[1] = 0; // Cmd Amp

			if((prc->Status == prcsSTATUS_Stopped) || prc->Disable){

				prc->Fbk[0] = 0.0;
				prc->Fbk[1] = (*HW_PS_Param_Set[i].pAmpSP);

			}else
				prc->Fbk[0] = prc->Fbk[1]; // cur Amp as  Cmd Amp

			// for implementation in future
			prc->Fbk[2] = 0; //varCurHW_Volt
			prc->Fbk[3] = 0; //varHW_Volt_Cmd

}

}
```

### Program Logical/Universal/ProgrTest

#### Cyclic.c
```c
#include <bur/plctypes.h>

#ifdef _DEFAULT_INCLUDES
	#include <AsDefault.h>
#endif

#include <..\..\Lib\utilityLib\bgdebug.h>
#include <..\..\Lib\ringbuffer\ringbuffer.h>
#include <..\..\Lib\ringbuffer\ringbuffer.c>

#include <..\..\Lib\arclink\arclink.h>
#include <..\..\Lib\arclink\arclink.c>

_LOCAL Arc_Link_typ *arcLink;
_LOCAL UDP_typ UDP;

void _INIT ProgramCyclic(void)
{UDP_typ *udp;

	udp = &UDP;

	udp->send.iBufferSize = RingBuffer_readRecord(arcLink->bufOUT, udp->send.iBuffer);

	Udp_cyclic(&UDP);
	DBG("Dupa");
	arcLink = 0;
}
```

Listed in the project but not available here: Logical/FourAxisTigCtrl/GlobDef.h, Logical/FourAxisTigCtrl/GlobDecl.h, Logical/FourAxisTigCtrl/HMI_Cntrl.c, Logical/FourAxisTigCtrl/PermSaving, Logical/FourAxisTigCtrl/AVC_SYNCH, Logical/FourAxisTigCtrl/HMI_M, Logical/Libraries/sprintf2/cvtflasc.c, Logical/Libraries/sprintf2/ofmt.c, Logical/Libraries/sprintf2/sprintf.c, Logical/Libraries/sprintf2/sprintf2.h
